LIN {X 0,Y 523.961,Z 128.215,A -85,B 0,C 180,E1 -4877.969,E2 -4877.969} C_VEL
LIN {X 0,Y 523.969,Z 128.221,A -85,B 0,C 180,E1 -4880.41,E2 -4880.41} C_VEL
LIN {X 0,Y 523.908,Z 128.222,A -85,B 0,C 180,E1 -4882.893,E2 -4882.893} C_VEL
LIN {X 0,Y 523.951,Z 128.214,A -85,B 0,C 180,E1 -4885.418,E2 -4885.418} C_VEL
LIN {X 0,Y 523.967,Z 128.217,A -85,B 0,C 180,E1 -4887.998,E2 -4887.998} C_VEL
LIN {X 0,Y 523.943,Z 128.216,A -85,B 0,C 180,E1 -4890.855,E2 -4890.855} C_VEL
LIN {X 0,Y 523.957,Z 128.217,A -85,B 0,C 180,E1 -4893.735,E2 -4893.735} C_VEL
LIN {X 0,Y 523.917,Z 128.223,A -85,B 0,C 180,E1 -4896.404,E2 -4896.404} C_VEL
LIN {X 0,Y 523.956,Z 128.214,A -85,B 0,C 180,E1 -4899.081,E2 -4899.081} C_VEL
LIN {X 0,Y 523.953,Z 128.221,A -85,B 0,C 180,E1 -4902.118,E2 -4902.118} C_VEL
LIN {X 0,Y 523.952,Z 128.216,A -85,B 0,C 180,E1 -4905.308,E2 -4905.308} C_VEL
LIN {X 0,Y 523.918,Z 128.218,A -85,B 0,C 180,E1 -4906.913,E2 -4906.913} C_VEL
LIN {X 0,Y 523.253,Z 128.307,A -85,B 0,C 180,E1 -4907.554,E2 -4907.554} C_VEL
LIN {X 0,Y 520.418,Z 128.661,A -85,B 0,C 180,E1 -4908.596,E2 -4908.596} C_VEL
LIN {X 0,Y 518.021,Z 128.96,A -85,B 0,C 180,E1 -4909.435,E2 -4909.435} C_VEL
LIN {X 0,Y 516.991,Z 129.087,A -85,B 0,C 180,E1 -4910.083,E2 -4910.083} C_VEL
LIN {X 0,Y 516.906,Z 129.094,A -85,B 0,C 180,E1 -4910.302,E2 -4910.302} C_VEL
LIN {X 0,Y 516.88,Z 129.098,A -85,B 0,C 180,E1 -4913.342,E2 -4913.342} C_VEL
LIN {X 0,Y 516.906,Z 129.095,A -85,B 0,C 180,E1 -4916.121,E2 -4916.121} C_VEL
LIN {X 0,Y 516.888,Z 129.095,A -85,B 0,C 180,E1 -4918.935,E2 -4918.935} C_VEL
LIN {X 0,Y 516.915,Z 129.1,A -85,B 0,C 180,E1 -4921.585,E2 -4921.585} C_VEL
LIN {X 0,Y 516.927,Z 129.09,A -85,B 0,C 180,E1 -4924.211,E2 -4924.211} C_VEL
LIN {X 0,Y 516.868,Z 129.097,A -85,B 0,C 180,E1 -4926.777,E2 -4926.777} C_VEL
LIN {X 0,Y 516.935,Z 129.093,A -85,B 0,C 180,E1 -4929.732,E2 -4929.732} C_VEL
LIN {X 0,Y 516.925,Z 129.09,A -85,B 0,C 180,E1 -4932.596,E2 -4932.596} C_VEL
LIN {X 0,Y 516.947,Z 129.092,A -85,B 0,C 180,E1 -4935.031,E2 -4935.031} C_VEL
LIN {X 0,Y 516.961,Z 129.085,A -85,B 0,C 180,E1 -4938.234,E2 -4938.234} C_VEL
LIN {X 0,Y 516.966,Z 129.09,A -85,B 0,C 180,E1 -4941.4,E2 -4941.4} C_VEL
LIN {X 0,Y 517.013,Z 129.08,A -85,B 0,C 180,E1 -4943.757,E2 -4943.757} C_VEL
LIN {X 0,Y 517.083,Z 129.071,A -85,B 0,C 180,E1 -4947.664,E2 -4947.664} C_VEL
LIN {X 0,Y 517.091,Z 129.075,A -85,B 0,C 180,E1 -4950.779,E2 -4950.779} C_VEL
LIN {X 0,Y 517.01,Z 129.085,A -85,B 0,C 180,E1 -4953.117,E2 -4953.117} C_VEL
LIN {X 0,Y 517.014,Z 129.08,A -85,B 0,C 180,E1 -4956.244,E2 -4956.244} C_VEL
LIN {X 0,Y 516.952,Z 129.088,A -85,B 0,C 180,E1 -4959.39,E2 -4959.39} C_VEL
LIN {X 0,Y 516.95,Z 129.086,A -85,B 0,C 180,E1 -4961.808,E2 -4961.808} C_VEL
LIN {X 0,Y 516.945,Z 129.092,A -85,B 0,C 180,E1 -4965.148,E2 -4965.148} C_VEL
LIN {X 0,Y 516.931,Z 129.096,A -85,B 0,C 180,E1 -4968.222,E2 -4968.222} C_VEL
LIN {X 0,Y 516.964,Z 129.166,A -85,B 0,C 180,E1 -4968.889,E2 -4968.889} C_VEL
LIN {X 0,Y 517.489,Z 133.922,A -85,B 0,C 180,E1 -4969.848,E2 -4969.848} C_VEL
LIN {X 0,Y 517.251,Z 148.414,A -85,B 0,C 180,E1 -4972.697,E2 -4972.697} C_VEL
LIN {X 0,Y 519.127,Z 158.271,A -85,B 0,C 180,E1 -4972.899,E2 -4972.899} C_VEL
LIN {X 0,Y 518.582,Z 255.219,A -85,B 0,C 180,E1 -4974.279,E2 -4974.279} C_VEL
LIN {X 0,Y 518.384,Z 268.208,A -85,B 0,C 180,E1 -4974.619,E2 -4974.619} C_VEL
LIN {X 0,Y 518.188,Z 281.309,A -85,B 0,C 180,E1 -4975.131,E2 -4975.131} C_VEL
LIN {X 0,Y 517.999,Z 292.599,A -85,B 0,C 180,E1 -4975.733,E2 -4975.733} C_VEL
LIN {X 0,Y 517.621,Z 304.359,A -85,B 0,C 180,E1 -4976.536,E2 -4976.536} C_VEL
LIN {X 0,Y 517.359,Z 314.43,A -85,B 0,C 180,E1 -4977.399,E2 -4977.399} C_VEL
LIN {X 0,Y 517.077,Z 323.966,A -85,B 0,C 180,E1 -4978.406,E2 -4978.406} C_VEL
LIN {X 0,Y 516.85,Z 332.431,A -85,B 0,C 180,E1 -4979.513,E2 -4979.513} C_VEL
LIN {X 0,Y 516.626,Z 340.432,A -85,B 0,C 180,E1 -4980.813,E2 -4980.813} C_VEL
LIN {X 0,Y 516.488,Z 346.396,A -85,B 0,C 180,E1 -4982.052,E2 -4982.052} C_VEL
LIN {X 0,Y 516.364,Z 351.459,A -85,B 0,C 180,E1 -4983.427,E2 -4983.427} C_VEL
LIN {X 0,Y 516.249,Z 355.267,A -85,B 0,C 180,E1 -4984.874,E2 -4984.874} C_VEL
LIN {X 0,Y 516.218,Z 356.939,A -85,B 0,C 180,E1 -4985.833,E2 -4985.833} C_VEL
LIN {X 0,Y 516.192,Z 358.058,A -85,B 0,C 180,E1 -4986.803,E2 -4986.803} C_VEL
LIN {X 0,Y 516.165,Z 358.528,A -85,B 0,C 180,E1 -4987.842,E2 -4987.842} C_VEL
LIN {X 0,Y 516.185,Z 358.189,A -85,B 0,C 180,E1 -4989.099,E2 -4989.099} C_VEL
LIN {X 0,Y 516.22,Z 356.867,A -85,B 0,C 180,E1 -4990.324,E2 -4990.324} C_VEL
LIN {X 0,Y 516.332,Z 353.874,A -85,B 0,C 180,E1 -4991.833,E2 -4991.833} C_VEL
LIN {X 0,Y 516.424,Z 349.132,A -85,B 0,C 180,E1 -4993.363,E2 -4993.363} C_VEL
LIN {X 0,Y 516.566,Z 343.421,A -85,B 0,C 180,E1 -4994.71,E2 -4994.71} C_VEL
LIN {X 0,Y 516.733,Z 337.42,A -85,B 0,C 180,E1 -4995.82,E2 -4995.82} C_VEL
LIN {X 0,Y 516.938,Z 329.156,A -85,B 0,C 180,E1 -4997.046,E2 -4997.046} C_VEL
LIN {X 0,Y 517.221,Z 320.09,A -85,B 0,C 180,E1 -4998.132,E2 -4998.132} C_VEL
LIN {X 0,Y 517.473,Z 310.551,A -85,B 0,C 180,E1 -4999.058,E2 -4999.058} C_VEL
LIN {X 0,Y 517.739,Z 300.481,A -85,B 0,C 180,E1 -4999.851,E2 -4999.851} C_VEL
LIN {X 0,Y 518.097,Z 289.313,A -85,B 0,C 180,E1 -5000.553,E2 -5000.553} C_VEL
LIN {X 0,Y 518.357,Z 276.664,A -85,B 0,C 180,E1 -5001.167,E2 -5001.167} C_VEL
LIN {X 0,Y 518.481,Z 264.053,A -85,B 0,C 180,E1 -5001.601,E2 -5001.601} C_VEL
LIN {X 0,Y 518.64,Z 250.833,A -85,B 0,C 180,E1 -5001.888,E2 -5001.888} C_VEL
LIN {X 0,Y 519.123,Z 157.894,A -85,B 0,C 180,E1 -5003.2,E2 -5003.2} C_VEL
LIN {X 0,Y 517.274,Z 148.573,A -85,B 0,C 180,E1 -5003.404,E2 -5003.404} C_VEL
LIN {X 0,Y 517.435,Z 134.125,A -85,B 0,C 180,E1 -5006.161,E2 -5006.161} C_VEL
LIN {X 0,Y 516.966,Z 129.093,A -85,B 0,C 180,E1 -5007.176,E2 -5007.176} C_VEL
LIN {X 0,Y 516.923,Z 129.093,A -85,B 0,C 180,E1 -5010.696,E2 -5010.696} C_VEL
LIN {X 0,Y 516.913,Z 129.096,A -85,B 0,C 180,E1 -5013.812,E2 -5013.812} C_VEL
LIN {X 0,Y 516.86,Z 129.105,A -85,B 0,C 180,E1 -5016.777,E2 -5016.777} C_VEL
LIN {X 0,Y 516.943,Z 129.09,A -85,B 0,C 180,E1 -5019.732,E2 -5019.732} C_VEL
LIN {X 0,Y 516.899,Z 129.099,A -85,B 0,C 180,E1 -5022.596,E2 -5022.596} C_VEL
LIN {X 0,Y 516.944,Z 129.095,A -85,B 0,C 180,E1 -5025.031,E2 -5025.031} C_VEL
LIN {X 0,Y 516.971,Z 129.089,A -85,B 0,C 180,E1 -5028.234,E2 -5028.234} C_VEL
LIN {X 0,Y 516.957,Z 129.088,A -85,B 0,C 180,E1 -5031.4,E2 -5031.4} C_VEL
LIN {X 0,Y 516.99,Z 129.089,A -85,B 0,C 180,E1 -5034.54,E2 -5034.54} C_VEL
LIN {X 0,Y 517.078,Z 129.073,A -85,B 0,C 180,E1 -5037.664,E2 -5037.664} C_VEL
LIN {X 0,Y 517.07,Z 129.075,A -85,B 0,C 180,E1 -5040,E2 -5040} C_VEL
LIN {X 0,Y 517.077,Z 129.075,A -85,B 0,C 180,E1 -5042.337,E2 -5042.337} C_VEL
LIN {X 0,Y 516.971,Z 129.086,A -85,B 0,C 180,E1 -5046.244,E2 -5046.244} C_VEL
LIN {X 0,Y 516.909,Z 129.094,A -85,B 0,C 180,E1 -5049.39,E2 -5049.39} C_VEL
LIN {X 0,Y 516.883,Z 129.095,A -85,B 0,C 180,E1 -5052.566,E2 -5052.566} C_VEL
LIN {X 0,Y 516.831,Z 129.107,A -85,B 0,C 180,E1 -5055.782,E2 -5055.782} C_VEL
LIN {X 0,Y 516.84,Z 129.101,A -85,B 0,C 180,E1 -5058.226,E2 -5058.226} C_VEL
LIN {X 0,Y 516.86,Z 129.098,A -85,B 0,C 180,E1 -5060.704,E2 -5060.704} C_VEL
LIN {X 0,Y 516.841,Z 129.107,A -85,B 0,C 180,E1 -5063.225,E2 -5063.225} C_VEL
LIN {X 0,Y 516.863,Z 129.098,A -85,B 0,C 180,E1 -5066.177,E2 -5066.177} C_VEL
LIN {X 0,Y 516.833,Z 129.1,A -85,B 0,C 180,E1 -5068.421,E2 -5068.421} C_VEL
LIN {X 0,Y 516.853,Z 129.105,A -85,B 0,C 180,E1 -5071.112,E2 -5071.112} C_VEL
LIN {X 0,Y 516.886,Z 129.095,A -85,B 0,C 180,E1 -5073.961,E2 -5073.961} C_VEL
LIN {X 0,Y 516.858,Z 129.105,A -85,B 0,C 180,E1 -5076.748,E2 -5076.748} C_VEL
LIN {X 0,Y 516.863,Z 129.099,A -85,B 0,C 180,E1 -5079.724,E2 -5079.724} C_VEL
LIN {X 0,Y 516.847,Z 129.107,A -85,B 0,C 180,E1 -5082.836,E2 -5082.836} C_VEL
LIN {X 0,Y 516.901,Z 129.098,A -85,B 0,C 180,E1 -5085.007,E2 -5085.007} C_VEL
LIN {X 0,Y 516.903,Z 129.102,A -85,B 0,C 180,E1 -5088.401,E2 -5088.401} C_VEL
LIN {X 0,Y 516.881,Z 129.097,A -85,B 0,C 180,E1 -5091.284,E2 -5091.284} C_VEL
LIN {X 0,Y 516.873,Z 129.105,A -85,B 0,C 180,E1 -5094.219,E2 -5094.219} C_VEL
LIN {X 0,Y 516.9,Z 129.097,A -85,B 0,C 180,E1 -5097.053,E2 -5097.053} C_VEL
LIN {X 0,Y 516.89,Z 129.102,A -85,B 0,C 180,E1 -5099.796,E2 -5099.796} C_VEL
LIN {X 0,Y 516.904,Z 129.098,A -85,B 0,C 180,E1 -5102.465,E2 -5102.465} C_VEL
LIN {X 0,Y 516.94,Z 129.172,A -85,B 0,C 180,E1 -5105.019,E2 -5105.019} C_VEL
LIN {X 0,Y 518.404,Z 137.817,A -85,B 0,C 180,E1 -5106.426,E2 -5106.426} C_VEL
LIN {X 0,Y 517.908,Z 158.298,A -85,B 0,C 180,E1 -5109.545,E2 -5109.545} C_VEL
LIN {X 0,Y 517.54,Z 177.537,A -85,B 0,C 180,E1 -5112.439,E2 -5112.439} C_VEL
LIN {X 0,Y 517.196,Z 192.388,A -85,B 0,C 180,E1 -5114.631,E2 -5114.631} C_VEL
LIN {X 0,Y 519.037,Z 206.215,A -85,B 0,C 180,E1 -5114.883,E2 -5114.883} C_VEL
LIN {X 0,Y 518.573,Z 300.986,A -85,B 0,C 180,E1 -5116.23,E2 -5116.23} C_VEL
LIN {X 0,Y 518.317,Z 314.244,A -85,B 0,C 180,E1 -5116.573,E2 -5116.573} C_VEL
LIN {X 0,Y 518.011,Z 326.993,A -85,B 0,C 180,E1 -5117.064,E2 -5117.064} C_VEL
LIN {X 0,Y 517.751,Z 338.84,A -85,B 0,C 180,E1 -5117.686,E2 -5117.686} C_VEL
LIN {X 0,Y 517.454,Z 350.053,A -85,B 0,C 180,E1 -5118.443,E2 -5118.443} C_VEL
LIN {X 0,Y 517.162,Z 360.598,A -85,B 0,C 180,E1 -5119.329,E2 -5119.329} C_VEL
LIN {X 0,Y 516.896,Z 369.22,A -85,B 0,C 180,E1 -5120.214,E2 -5120.214} C_VEL
LIN {X 0,Y 516.68,Z 377.176,A -85,B 0,C 180,E1 -5121.197,E2 -5121.197} C_VEL
LIN {X 0,Y 516.516,Z 384.949,A -85,B 0,C 180,E1 -5122.376,E2 -5122.376} C_VEL
LIN {X 0,Y 516.376,Z 392.107,A -85,B 0,C 180,E1 -5123.749,E2 -5123.749} C_VEL
LIN {X 0,Y 516.312,Z 396.873,A -85,B 0,C 180,E1 -5124.924,E2 -5124.924} C_VEL
LIN {X 0,Y 516.352,Z 400.52,A -85,B 0,C 180,E1 -5126.097,E2 -5126.097} C_VEL
LIN {X 0,Y 516.303,Z 402.399,A -85,B 0,C 180,E1 -5126.878,E2 -5126.878} C_VEL
LIN {X 0,Y 516.264,Z 403.807,A -85,B 0,C 180,E1 -5127.659,E2 -5127.659} C_VEL
LIN {X 0,Y 516.172,Z 405.428,A -85,B 0,C 180,E1 -5129.219,E2 -5129.219} C_VEL
LIN {X 0,Y 516.173,Z 405.651,A -85,B 0,C 180,E1 -5130,E2 -5130} C_VEL
LIN {X 0,Y 516.193,Z 404.83,A -85,B 0,C 180,E1 -5131.56,E2 -5131.56} C_VEL
LIN {X 0,Y 516.264,Z 403.836,A -85,B 0,C 180,E1 -5132.34,E2 -5132.34} C_VEL
LIN {X 0,Y 516.303,Z 402.435,A -85,B 0,C 180,E1 -5133.121,E2 -5133.121} C_VEL
LIN {X 0,Y 516.31,Z 399.485,A -85,B 0,C 180,E1 -5134.293,E2 -5134.293} C_VEL
LIN {X 0,Y 516.367,Z 395.491,A -85,B 0,C 180,E1 -5135.467,E2 -5135.467} C_VEL
LIN {X 0,Y 516.41,Z 390.303,A -85,B 0,C 180,E1 -5136.651,E2 -5136.651} C_VEL
LIN {X 0,Y 516.534,Z 383.867,A -85,B 0,C 180,E1 -5137.82,E2 -5137.82} C_VEL
LIN {X 0,Y 516.741,Z 375.791,A -85,B 0,C 180,E1 -5138.998,E2 -5138.998} C_VEL
LIN {X 0,Y 516.93,Z 367.556,A -85,B 0,C 180,E1 -5139.982,E2 -5139.982} C_VEL
LIN {X 0,Y 517.224,Z 357.517,A -85,B 0,C 180,E1 -5140.966,E2 -5140.966} C_VEL
LIN {X 0,Y 517.504,Z 347.593,A -85,B 0,C 180,E1 -5141.753,E2 -5141.753} C_VEL
LIN {X 0,Y 517.83,Z 336.445,A -85,B 0,C 180,E1 -5142.462,E2 -5142.462} C_VEL
LIN {X 0,Y 518.108,Z 323.829,A -85,B 0,C 180,E1 -5143.083,E2 -5143.083} C_VEL
LIN {X 0,Y 518.408,Z 311.414,A -85,B 0,C 180,E1 -5143.524,E2 -5143.524} C_VEL
LIN {X 0,Y 518.607,Z 298.558,A -85,B 0,C 180,E1 -5143.818,E2 -5143.818} C_VEL
LIN {X 0,Y 518.962,Z 204.412,A -85,B 0,C 180,E1 -5145.149,E2 -5145.149} C_VEL
LIN {X 0,Y 517.228,Z 192.469,A -85,B 0,C 180,E1 -5145.389,E2 -5145.389} C_VEL
LIN {X 0,Y 517.694,Z 172.47,A -85,B 0,C 180,E1 -5148.399,E2 -5148.399} C_VEL
LIN {X 0,Y 518.188,Z 152.265,A -85,B 0,C 180,E1 -5151.48,E2 -5151.48} C_VEL
LIN {X 0,Y 518.583,Z 138.788,A -85,B 0,C 180,E1 -5153.565,E2 -5153.565} C_VEL
LIN {X 0,Y 517.236,Z 130.625,A -85,B 0,C 180,E1 -5154.911,E2 -5154.911} C_VEL
LIN {X 0,Y 516.922,Z 129.096,A -85,B 0,C 180,E1 -5155.196,E2 -5155.196} C_VEL
LIN {X 0,Y 516.917,Z 129.098,A -85,B 0,C 180,E1 -5157.903,E2 -5157.903} C_VEL
LIN {X 0,Y 516.893,Z 129.101,A -85,B 0,C 180,E1 -5160.203,E2 -5160.203} C_VEL
LIN {X 0,Y 516.896,Z 129.093,A -85,B 0,C 180,E1 -5162.946,E2 -5162.946} C_VEL
LIN {X 0,Y 516.871,Z 129.103,A -85,B 0,C 180,E1 -5165.78,E2 -5165.78} C_VEL
LIN {X 0,Y 516.882,Z 129.095,A -85,B 0,C 180,E1 -5168.715,E2 -5168.715} C_VEL
LIN {X 0,Y 516.912,Z 129.099,A -85,B 0,C 180,E1 -5171.775,E2 -5171.775} C_VEL
LIN {X 0,Y 516.895,Z 129.094,A -85,B 0,C 180,E1 -5175.006,E2 -5175.006} C_VEL
LIN {X 0,Y 516.915,Z 129.091,A -85,B 0,C 180,E1 -5178.398,E2 -5178.398} C_VEL
LIN {X 0,Y 516.88,Z 129.099,A -85,B 0,C 180,E1 -5181.284,E2 -5181.284} C_VEL
LIN {X 0,Y 516.87,Z 129.097,A -85,B 0,C 180,E1 -5184.219,E2 -5184.219} C_VEL
LIN {X 0,Y 516.88,Z 129.098,A -85,B 0,C 180,E1 -5187.052,E2 -5187.052} C_VEL
LIN {X 0,Y 516.886,Z 129.098,A -85,B 0,C 180,E1 -5189.796,E2 -5189.796} C_VEL
LIN {X 0,Y 516.925,Z 129.089,A -85,B 0,C 180,E1 -5192.467,E2 -5192.467} C_VEL
LIN {X 0,Y 516.908,Z 129.096,A -85,B 0,C 180,E1 -5195.071,E2 -5195.071} C_VEL
LIN {X 0,Y 516.885,Z 129.095,A -85,B 0,C 180,E1 -5198.462,E2 -5198.462} C_VEL
LIN {X 0,Y 516.899,Z 129.098,A -85,B 0,C 180,E1 -5200.954,E2 -5200.954} C_VEL
LIN {X 0,Y 516.907,Z 129.097,A -85,B 0,C 180,E1 -5203.41,E2 -5203.41} C_VEL
LIN {X 0,Y 516.893,Z 129.094,A -85,B 0,C 180,E1 -5205.833,E2 -5205.833} C_VEL
LIN {X 0,Y 516.965,Z 129.085,A -85,B 0,C 180,E1 -5208.233,E2 -5208.233} C_VEL
LIN {X 0,Y 516.967,Z 129.088,A -85,B 0,C 180,E1 -5211.399,E2 -5211.399} C_VEL
LIN {X 0,Y 517.002,Z 129.08,A -85,B 0,C 180,E1 -5213.756,E2 -5213.756} C_VEL
LIN {X 0,Y 517.012,Z 129.088,A -85,B 0,C 180,E1 -5216.883,E2 -5216.883} C_VEL
LIN {X 0,Y 517.084,Z 129.07,A -85,B 0,C 180,E1 -5220,E2 -5220} C_VEL
LIN {X 0,Y 517.01,Z 129.083,A -85,B 0,C 180,E1 -5223.117,E2 -5223.117} C_VEL
LIN {X 0,Y 517.001,Z 129.083,A -85,B 0,C 180,E1 -5226.243,E2 -5226.243} C_VEL
LIN {X 0,Y 516.952,Z 129.087,A -85,B 0,C 180,E1 -5229.389,E2 -5229.389} C_VEL
LIN {X 0,Y 516.95,Z 129.087,A -85,B 0,C 180,E1 -5231.807,E2 -5231.807} C_VEL
LIN {X 0,Y 516.944,Z 129.088,A -85,B 0,C 180,E1 -5235.147,E2 -5235.147} C_VEL
LIN {X 0,Y 516.922,Z 129.095,A -85,B 0,C 180,E1 -5238.222,E2 -5238.222} C_VEL
LIN {X 0,Y 516.909,Z 129.096,A -85,B 0,C 180,E1 -5240.701,E2 -5240.701} C_VEL
LIN {X 0,Y 516.9,Z 129.097,A -85,B 0,C 180,E1 -5244.072,E2 -5244.072} C_VEL
LIN {X 0,Y 516.926,Z 129.093,A -85,B 0,C 180,E1 -5246.657,E2 -5246.657} C_VEL
LIN {X 0,Y 516.908,Z 129.092,A -85,B 0,C 180,E1 -5249.524,E2 -5249.524} C_VEL
LIN {X 0,Y 516.897,Z 129.097,A -85,B 0,C 180,E1 -5252.544,E2 -5252.544} C_VEL
LIN {X 0,Y 516.876,Z 129.096,A -85,B 0,C 180,E1 -5255.332,E2 -5255.332} C_VEL
LIN {X 0,Y 516.878,Z 129.103,A -85,B 0,C 180,E1 -5257.943,E2 -5257.943} C_VEL
LIN {X 0,Y 516.9,Z 129.093,A -85,B 0,C 180,E1 -5260.739,E2 -5260.739} C_VEL
LIN {X 0,Y 516.878,Z 129.104,A -85,B 0,C 180,E1 -5263.903,E2 -5263.903} C_VEL
LIN {X 0,Y 516.878,Z 129.101,A -85,B 0,C 180,E1 -5266.107,E2 -5266.107} C_VEL
LIN {X 0,Y 516.899,Z 129.094,A -85,B 0,C 180,E1 -5269.26,E2 -5269.26} C_VEL
LIN {X 0,Y 516.906,Z 129.094,A -85,B 0,C 180,E1 -5270.302,E2 -5270.302} C_VEL
LIN {X 0,Y 516.237,Z 129.176,A -85,B 0,C 180,E1 -5270.952,E2 -5270.952} C_VEL
LIN {X 0,Y 513.38,Z 129.538,A -85,B 0,C 180,E1 -5272.007,E2 -5272.007} C_VEL
LIN {X 0,Y 510.961,Z 129.844,A -85,B 0,C 180,E1 -5272.857,E2 -5272.857} C_VEL
LIN {X 0,Y 509.915,Z 129.972,A -85,B 0,C 180,E1 -5273.514,E2 -5273.514} C_VEL
LIN {X 0,Y 509.826,Z 129.98,A -85,B 0,C 180,E1 -5273.736,E2 -5273.736} C_VEL
LIN {X 0,Y 509.857,Z 129.97,A -85,B 0,C 180,E1 -5276.539,E2 -5276.539} C_VEL
LIN {X 0,Y 509.841,Z 129.976,A -85,B 0,C 180,E1 -5279.334,E2 -5279.334} C_VEL
LIN {X 0,Y 509.89,Z 129.968,A -85,B 0,C 180,E1 -5282.055,E2 -5282.055} C_VEL
LIN {X 0,Y 509.873,Z 129.968,A -85,B 0,C 180,E1 -5284.704,E2 -5284.704} C_VEL
LIN {X 0,Y 509.852,Z 129.98,A -85,B 0,C 180,E1 -5287.45,E2 -5287.45} C_VEL
LIN {X 0,Y 509.913,Z 129.966,A -85,B 0,C 180,E1 -5289.845,E2 -5289.845} C_VEL
LIN {X 0,Y 509.881,Z 129.973,A -85,B 0,C 180,E1 -5293.175,E2 -5293.175} C_VEL
LIN {X 0,Y 509.869,Z 129.972,A -85,B 0,C 180,E1 -5295.635,E2 -5295.635} C_VEL
LIN {X 0,Y 509.91,Z 129.967,A -85,B 0,C 180,E1 -5298.875,E2 -5298.875} C_VEL
LIN {X 0,Y 509.948,Z 129.959,A -85,B 0,C 180,E1 -5302.079,E2 -5302.079} C_VEL
LIN {X 0,Y 509.983,Z 129.955,A -85,B 0,C 180,E1 -5304.465,E2 -5304.465} C_VEL
LIN {X 0,Y 510.054,Z 129.947,A -85,B 0,C 180,E1 -5307.631,E2 -5307.631} C_VEL
LIN {X 0,Y 510.061,Z 129.951,A -85,B 0,C 180,E1 -5310.79,E2 -5310.79} C_VEL
LIN {X 0,Y 509.952,Z 129.964,A -85,B 0,C 180,E1 -5313.161,E2 -5313.161} C_VEL
LIN {X 0,Y 509.981,Z 129.956,A -85,B 0,C 180,E1 -5316.33,E2 -5316.33} C_VEL
LIN {X 0,Y 509.914,Z 129.97,A -85,B 0,C 180,E1 -5318.721,E2 -5318.721} C_VEL
LIN {X 0,Y 509.902,Z 129.965,A -85,B 0,C 180,E1 -5321.932,E2 -5321.932} C_VEL
LIN {X 0,Y 509.892,Z 129.97,A -85,B 0,C 180,E1 -5325.242,E2 -5325.242} C_VEL
LIN {X 0,Y 509.883,Z 129.976,A -85,B 0,C 180,E1 -5328.483,E2 -5328.483} C_VEL
LIN {X 0,Y 509.945,Z 130.203,A -85,B 0,C 180,E1 -5328.794,E2 -5328.794} C_VEL
LIN {X 0,Y 510.5,Z 135.748,A -85,B 0,C 180,E1 -5329.922,E2 -5329.922} C_VEL
LIN {X 0,Y 510.268,Z 148.653,A -85,B 0,C 180,E1 -5332.48,E2 -5332.48} C_VEL
LIN {X 0,Y 512.304,Z 159.447,A -85,B 0,C 180,E1 -5332.706,E2 -5332.706} C_VEL
LIN {X 0,Y 511.687,Z 256.025,A -85,B 0,C 180,E1 -5334.105,E2 -5334.105} C_VEL
LIN {X 0,Y 511.49,Z 269.228,A -85,B 0,C 180,E1 -5334.462,E2 -5334.462} C_VEL
LIN {X 0,Y 511.297,Z 281.411,A -85,B 0,C 180,E1 -5334.948,E2 -5334.948} C_VEL
LIN {X 0,Y 511.071,Z 292.81,A -85,B 0,C 180,E1 -5335.56,E2 -5335.56} C_VEL
LIN {X 0,Y 510.738,Z 303.116,A -85,B 0,C 180,E1 -5336.261,E2 -5336.261} C_VEL
LIN {X 0,Y 510.416,Z 313.477,A -85,B 0,C 180,E1 -5337.136,E2 -5337.136} C_VEL
LIN {X 0,Y 510.097,Z 323.155,A -85,B 0,C 180,E1 -5338.144,E2 -5338.144} C_VEL
LIN {X 0,Y 509.847,Z 332.075,A -85,B 0,C 180,E1 -5339.298,E2 -5339.298} C_VEL
LIN {X 0,Y 509.636,Z 339.27,A -85,B 0,C 180,E1 -5340.451,E2 -5340.451} C_VEL
LIN {X 0,Y 509.461,Z 345.149,A -85,B 0,C 180,E1 -5341.616,E2 -5341.616} C_VEL
LIN {X 0,Y 509.307,Z 350.833,A -85,B 0,C 180,E1 -5343.063,E2 -5343.063} C_VEL
LIN {X 0,Y 509.203,Z 354.759,A -85,B 0,C 180,E1 -5344.464,E2 -5344.464} C_VEL
LIN {X 0,Y 509.132,Z 356.774,A -85,B 0,C 180,E1 -5345.47,E2 -5345.47} C_VEL
LIN {X 0,Y 509.1,Z 358.394,A -85,B 0,C 180,E1 -5346.806,E2 -5346.806} C_VEL
LIN {X 0,Y 509.083,Z 358.882,A -85,B 0,C 180,E1 -5348.104,E2 -5348.104} C_VEL
LIN {X 0,Y 509.114,Z 358.288,A -85,B 0,C 180,E1 -5349.421,E2 -5349.421} C_VEL
LIN {X 0,Y 509.156,Z 356.823,A -85,B 0,C 180,E1 -5350.609,E2 -5350.609} C_VEL
LIN {X 0,Y 509.263,Z 354.358,A -85,B 0,C 180,E1 -5351.823,E2 -5351.823} C_VEL
LIN {X 0,Y 509.345,Z 350.01,A -85,B 0,C 180,E1 -5353.28,E2 -5353.28} C_VEL
LIN {X 0,Y 509.495,Z 344.178,A -85,B 0,C 180,E1 -5354.709,E2 -5354.709} C_VEL
LIN {X 0,Y 509.68,Z 338.416,A -85,B 0,C 180,E1 -5355.811,E2 -5355.811} C_VEL
LIN {X 0,Y 509.854,Z 331.216,A -85,B 0,C 180,E1 -5356.935,E2 -5356.935} C_VEL
LIN {X 0,Y 510.159,Z 322.216,A -85,B 0,C 180,E1 -5358.066,E2 -5358.066} C_VEL
LIN {X 0,Y 510.486,Z 311.835,A -85,B 0,C 180,E1 -5359.121,E2 -5359.121} C_VEL
LIN {X 0,Y 510.763,Z 301.309,A -85,B 0,C 180,E1 -5359.976,E2 -5359.976} C_VEL
LIN {X 0,Y 511.141,Z 290.511,A -85,B 0,C 180,E1 -5360.674,E2 -5360.674} C_VEL
LIN {X 0,Y 511.403,Z 278.832,A -85,B 0,C 180,E1 -5361.263,E2 -5361.263} C_VEL
LIN {X 0,Y 511.58,Z 266.201,A -85,B 0,C 180,E1 -5361.732,E2 -5361.732} C_VEL
LIN {X 0,Y 511.718,Z 253.647,A -85,B 0,C 180,E1 -5362.034,E2 -5362.034} C_VEL
LIN {X 0,Y 512.294,Z 158.765,A -85,B 0,C 180,E1 -5363.4,E2 -5363.4} C_VEL
LIN {X 0,Y 510.314,Z 148.809,A -85,B 0,C 180,E1 -5363.631,E2 -5363.631} C_VEL
LIN {X 0,Y 510.453,Z 134.587,A -85,B 0,C 180,E1 -5366.361,E2 -5366.361} C_VEL
LIN {X 0,Y 509.906,Z 129.973,A -85,B 0,C 180,E1 -5367.292,E2 -5367.292} C_VEL
LIN {X 0,Y 509.86,Z 129.972,A -85,B 0,C 180,E1 -5370.275,E2 -5370.275} C_VEL
LIN {X 0,Y 509.878,Z 129.975,A -85,B 0,C 180,E1 -5372.945,E2 -5372.945} C_VEL
LIN {X 0,Y 509.843,Z 129.978,A -85,B 0,C 180,E1 -5375.573,E2 -5375.573} C_VEL
LIN {X 0,Y 509.824,Z 129.977,A -85,B 0,C 180,E1 -5378.149,E2 -5378.149} C_VEL
LIN {X 0,Y 509.86,Z 129.976,A -85,B 0,C 180,E1 -5380.682,E2 -5380.682} C_VEL
LIN {X 0,Y 509.867,Z 129.975,A -85,B 0,C 180,E1 -5383.175,E2 -5383.175} C_VEL
LIN {X 0,Y 509.858,Z 129.973,A -85,B 0,C 180,E1 -5385.634,E2 -5385.634} C_VEL
LIN {X 0,Y 509.916,Z 129.969,A -85,B 0,C 180,E1 -5388.875,E2 -5388.875} C_VEL
LIN {X 0,Y 509.912,Z 129.968,A -85,B 0,C 180,E1 -5392.078,E2 -5392.078} C_VEL
LIN {X 0,Y 509.945,Z 129.968,A -85,B 0,C 180,E1 -5394.464,E2 -5394.464} C_VEL
LIN {X 0,Y 510.046,Z 129.949,A -85,B 0,C 180,E1 -5397.631,E2 -5397.631} C_VEL
LIN {X 0,Y 510.038,Z 129.951,A -85,B 0,C 180,E1 -5400,E2 -5400} C_VEL
LIN {X 0,Y 510.045,Z 129.95,A -85,B 0,C 180,E1 -5402.37,E2 -5402.37} C_VEL
LIN {X 0,Y 509.939,Z 129.963,A -85,B 0,C 180,E1 -5405.537,E2 -5405.537} C_VEL
LIN {X 0,Y 509.879,Z 129.973,A -85,B 0,C 180,E1 -5407.923,E2 -5407.923} C_VEL
LIN {X 0,Y 509.864,Z 129.967,A -85,B 0,C 180,E1 -5411.127,E2 -5411.127} C_VEL
LIN {X 0,Y 509.815,Z 129.981,A -85,B 0,C 180,E1 -5413.554,E2 -5413.554} C_VEL
LIN {X 0,Y 509.792,Z 129.982,A -85,B 0,C 180,E1 -5416.005,E2 -5416.005} C_VEL
LIN {X 0,Y 509.806,Z 129.976,A -85,B 0,C 180,E1 -5418.486,E2 -5418.486} C_VEL
LIN {X 0,Y 509.812,Z 129.978,A -85,B 0,C 180,E1 -5421.004,E2 -5421.004} C_VEL
LIN {X 0,Y 509.802,Z 129.981,A -85,B 0,C 180,E1 -5423.565,E2 -5423.565} C_VEL
LIN {X 0,Y 509.804,Z 129.977,A -85,B 0,C 180,E1 -5426.353,E2 -5426.353} C_VEL
LIN {X 0,Y 509.797,Z 129.98,A -85,B 0,C 180,E1 -5428.85,E2 -5428.85} C_VEL
LIN {X 0,Y 509.801,Z 129.979,A -85,B 0,C 180,E1 -5431.592,E2 -5431.592} C_VEL
LIN {X 0,Y 509.839,Z 129.975,A -85,B 0,C 180,E1 -5434.415,E2 -5434.415} C_VEL
LIN {X 0,Y 509.812,Z 129.978,A -85,B 0,C 180,E1 -5437.342,E2 -5437.342} C_VEL
LIN {X 0,Y 509.819,Z 129.979,A -85,B 0,C 180,E1 -5440.385,E2 -5440.385} C_VEL
LIN {X 0,Y 509.81,Z 129.977,A -85,B 0,C 180,E1 -5443.573,E2 -5443.573} C_VEL
LIN {X 0,Y 509.813,Z 129.984,A -85,B 0,C 180,E1 -5446.427,E2 -5446.427} C_VEL
LIN {X 0,Y 509.826,Z 129.977,A -85,B 0,C 180,E1 -5449.305,E2 -5449.305} C_VEL
LIN {X 0,Y 509.854,Z 129.974,A -85,B 0,C 180,E1 -5451.787,E2 -5451.787} C_VEL
LIN {X 0,Y 509.832,Z 129.978,A -85,B 0,C 180,E1 -5454.622,E2 -5454.622} C_VEL
LIN {X 0,Y 509.866,Z 129.974,A -85,B 0,C 180,E1 -5457.481,E2 -5457.481} C_VEL
LIN {X 0,Y 509.863,Z 129.977,A -85,B 0,C 180,E1 -5460.274,E2 -5460.274} C_VEL
LIN {X 0,Y 509.884,Z 129.974,A -85,B 0,C 180,E1 -5463.629,E2 -5463.629} C_VEL
LIN {X 0,Y 509.888,Z 129.999,A -85,B 0,C 180,E1 -5464.838,E2 -5464.838} C_VEL
LIN {X 0,Y 511.457,Z 138.841,A -85,B 0,C 180,E1 -5466.301,E2 -5466.301} C_VEL
LIN {X 0,Y 510.986,Z 158.737,A -85,B 0,C 180,E1 -5469.378,E2 -5469.378} C_VEL
LIN {X 0,Y 510.526,Z 178.372,A -85,B 0,C 180,E1 -5472.37,E2 -5472.37} C_VEL
LIN {X 0,Y 510.198,Z 191.955,A -85,B 0,C 180,E1 -5474.413,E2 -5474.413} C_VEL
LIN {X 0,Y 512.182,Z 206.713,A -85,B 0,C 180,E1 -5474.689,E2 -5474.689} C_VEL
LIN {X 0,Y 511.683,Z 300.481,A -85,B 0,C 180,E1 -5476.041,E2 -5476.041} C_VEL
LIN {X 0,Y 511.395,Z 313.787,A -85,B 0,C 180,E1 -5476.388,E2 -5476.388} C_VEL
LIN {X 0,Y 511.071,Z 326.562,A -85,B 0,C 180,E1 -5476.885,E2 -5476.885} C_VEL
LIN {X 0,Y 510.77,Z 338.533,A -85,B 0,C 180,E1 -5477.521,E2 -5477.521} C_VEL
LIN {X 0,Y 510.448,Z 349.663,A -85,B 0,C 180,E1 -5478.282,E2 -5478.282} C_VEL
LIN {X 0,Y 510.15,Z 360.22,A -85,B 0,C 180,E1 -5479.181,E2 -5479.181} C_VEL
LIN {X 0,Y 509.835,Z 368.849,A -85,B 0,C 180,E1 -5480.077,E2 -5480.077} C_VEL
LIN {X 0,Y 509.64,Z 376.815,A -85,B 0,C 180,E1 -5481.075,E2 -5481.075} C_VEL
LIN {X 0,Y 509.429,Z 384.596,A -85,B 0,C 180,E1 -5482.269,E2 -5482.269} C_VEL
LIN {X 0,Y 509.31,Z 390.938,A -85,B 0,C 180,E1 -5483.483,E2 -5483.483} C_VEL
LIN {X 0,Y 509.241,Z 396.536,A -85,B 0,C 180,E1 -5484.853,E2 -5484.853} C_VEL
LIN {X 0,Y 509.246,Z 400.186,A -85,B 0,C 180,E1 -5486.043,E2 -5486.043} C_VEL
LIN {X 0,Y 509.219,Z 402.069,A -85,B 0,C 180,E1 -5486.835,E2 -5486.835} C_VEL
LIN {X 0,Y 509.193,Z 403.48,A -85,B 0,C 180,E1 -5487.626,E2 -5487.626} C_VEL
LIN {X 0,Y 509.085,Z 405.104,A -85,B 0,C 180,E1 -5489.209,E2 -5489.209} C_VEL
LIN {X 0,Y 509.083,Z 405.328,A -85,B 0,C 180,E1 -5490,E2 -5490} C_VEL
LIN {X 0,Y 509.113,Z 404.509,A -85,B 0,C 180,E1 -5491.582,E2 -5491.582} C_VEL
LIN {X 0,Y 509.193,Z 403.514,A -85,B 0,C 180,E1 -5492.373,E2 -5492.373} C_VEL
LIN {X 0,Y 509.219,Z 402.112,A -85,B 0,C 180,E1 -5493.164,E2 -5493.164} C_VEL
LIN {X 0,Y 509.203,Z 399.16,A -85,B 0,C 180,E1 -5494.353,E2 -5494.353} C_VEL
LIN {X 0,Y 509.279,Z 395.164,A -85,B 0,C 180,E1 -5495.543,E2 -5495.543} C_VEL
LIN {X 0,Y 509.366,Z 389.113,A -85,B 0,C 180,E1 -5496.914,E2 -5496.914} C_VEL
LIN {X 0,Y 509.493,Z 382.289,A -85,B 0,C 180,E1 -5498.128,E2 -5498.128} C_VEL
LIN {X 0,Y 509.715,Z 373.952,A -85,B 0,C 180,E1 -5499.323,E2 -5499.323} C_VEL
LIN {X 0,Y 509.957,Z 365.393,A -85,B 0,C 180,E1 -5500.32,E2 -5500.32} C_VEL
LIN {X 0,Y 510.328,Z 354.826,A -85,B 0,C 180,E1 -5501.317,E2 -5501.317} C_VEL
LIN {X 0,Y 510.584,Z 344.031,A -85,B 0,C 180,E1 -5502.14,E2 -5502.14} C_VEL
LIN {X 0,Y 510.934,Z 332.88,A -85,B 0,C 180,E1 -5502.814,E2 -5502.814} C_VEL
LIN {X 0,Y 511.218,Z 321.009,A -85,B 0,C 180,E1 -5503.363,E2 -5503.363} C_VEL
LIN {X 0,Y 511.529,Z 307.326,A -85,B 0,C 180,E1 -5503.81,E2 -5503.81} C_VEL
LIN {X 0,Y 511.754,Z 295.057,A -85,B 0,C 180,E1 -5504.058,E2 -5504.058} C_VEL
LIN {X 0,Y 511.999,Z 204.354,A -85,B 0,C 180,E1 -5505.356,E2 -5505.356} C_VEL
LIN {X 0,Y 510.208,Z 192.178,A -85,B 0,C 180,E1 -5505.603,E2 -5505.603} C_VEL
LIN {X 0,Y 510.752,Z 170.815,A -85,B 0,C 180,E1 -5508.866,E2 -5508.866} C_VEL
LIN {X 0,Y 511.358,Z 149.282,A -85,B 0,C 180,E1 -5512.207,E2 -5512.207} C_VEL
LIN {X 0,Y 511.528,Z 138.482,A -85,B 0,C 180,E1 -5513.91,E2 -5513.91} C_VEL
LIN {X 0,Y 509.874,Z 129.975,A -85,B 0,C 180,E1 -5515.35,E2 -5515.35} C_VEL
LIN {X 0,Y 509.89,Z 129.974,A -85,B 0,C 180,E1 -5518.098,E2 -5518.098} C_VEL
LIN {X 0,Y 509.847,Z 129.972,A -85,B 0,C 180,E1 -5521.279,E2 -5521.279} C_VEL
LIN {X 0,Y 509.857,Z 129.976,A -85,B 0,C 180,E1 -5524.202,E2 -5524.202} C_VEL
LIN {X 0,Y 509.817,Z 129.976,A -85,B 0,C 180,E1 -5527.34,E2 -5527.34} C_VEL
LIN {X 0,Y 509.838,Z 129.974,A -85,B 0,C 180,E1 -5530.382,E2 -5530.382} C_VEL
LIN {X 0,Y 509.822,Z 129.975,A -85,B 0,C 180,E1 -5533.062,E2 -5533.062} C_VEL
LIN {X 0,Y 509.823,Z 129.983,A -85,B 0,C 180,E1 -5535.793,E2 -5535.793} C_VEL
LIN {X 0,Y 509.857,Z 129.97,A -85,B 0,C 180,E1 -5538.574,E2 -5538.574} C_VEL
LIN {X 0,Y 509.851,Z 129.977,A -85,B 0,C 180,E1 -5541.786,E2 -5541.786} C_VEL
LIN {X 0,Y 509.829,Z 129.973,A -85,B 0,C 180,E1 -5544.621,E2 -5544.621} C_VEL
LIN {X 0,Y 509.859,Z 129.978,A -85,B 0,C 180,E1 -5547.48,E2 -5547.48} C_VEL
LIN {X 0,Y 509.857,Z 129.97,A -85,B 0,C 180,E1 -5550.273,E2 -5550.273} C_VEL
LIN {X 0,Y 509.883,Z 129.969,A -85,B 0,C 180,E1 -5552.944,E2 -5552.944} C_VEL
LIN {X 0,Y 509.864,Z 129.975,A -85,B 0,C 180,E1 -5555.573,E2 -5555.573} C_VEL
LIN {X 0,Y 509.849,Z 129.976,A -85,B 0,C 180,E1 -5558.998,E2 -5558.998} C_VEL
LIN {X 0,Y 509.86,Z 129.974,A -85,B 0,C 180,E1 -5561.516,E2 -5561.516} C_VEL
LIN {X 0,Y 509.852,Z 129.971,A -85,B 0,C 180,E1 -5563.997,E2 -5563.997} C_VEL
LIN {X 0,Y 509.861,Z 129.97,A -85,B 0,C 180,E1 -5566.447,E2 -5566.447} C_VEL
LIN {X 0,Y 509.912,Z 129.969,A -85,B 0,C 180,E1 -5568.874,E2 -5568.874} C_VEL
LIN {X 0,Y 509.95,Z 129.958,A -85,B 0,C 180,E1 -5572.078,E2 -5572.078} C_VEL
LIN {X 0,Y 509.979,Z 129.957,A -85,B 0,C 180,E1 -5574.464,E2 -5574.464} C_VEL
LIN {X 0,Y 510.055,Z 129.946,A -85,B 0,C 180,E1 -5577.63,E2 -5577.63} C_VEL
LIN {X 0,Y 510.063,Z 129.953,A -85,B 0,C 180,E1 -5580.789,E2 -5580.789} C_VEL
LIN {X 0,Y 509.952,Z 129.962,A -85,B 0,C 180,E1 -5583.16,E2 -5583.16} C_VEL
LIN {X 0,Y 509.953,Z 129.962,A -85,B 0,C 180,E1 -5586.329,E2 -5586.329} C_VEL
LIN {X 0,Y 509.914,Z 129.971,A -85,B 0,C 180,E1 -5588.72,E2 -5588.72} C_VEL
LIN {X 0,Y 509.902,Z 129.965,A -85,B 0,C 180,E1 -5591.931,E2 -5591.931} C_VEL
LIN {X 0,Y 509.891,Z 129.966,A -85,B 0,C 180,E1 -5595.241,E2 -5595.241} C_VEL
LIN {X 0,Y 509.886,Z 129.969,A -85,B 0,C 180,E1 -5598.001,E2 -5598.001} C_VEL
LIN {X 0,Y 509.847,Z 129.973,A -85,B 0,C 180,E1 -5601.001,E2 -5601.001} C_VEL
LIN {X 0,Y 509.862,Z 129.977,A -85,B 0,C 180,E1 -5604.426,E2 -5604.426} C_VEL
LIN {X 0,Y 509.884,Z 129.967,A -85,B 0,C 180,E1 -5607.055,E2 -5607.055} C_VEL
LIN {X 0,Y 509.853,Z 129.973,A -85,B 0,C 180,E1 -5609.751,E2 -5609.751} C_VEL
LIN {X 0,Y 509.873,Z 129.969,A -85,B 0,C 180,E1 -5612.775,E2 -5612.775} C_VEL
LIN {X 0,Y 509.836,Z 129.975,A -85,B 0,C 180,E1 -5615.581,E2 -5615.581} C_VEL
LIN {X 0,Y 509.855,Z 129.975,A -85,B 0,C 180,E1 -5618.337,E2 -5618.337} C_VEL
LIN {X 0,Y 509.861,Z 129.971,A -85,B 0,C 180,E1 -5621.424,E2 -5621.424} C_VEL
LIN {X 0,Y 509.852,Z 129.971,A -85,B 0,C 180,E1 -5624.668,E2 -5624.668} C_VEL
LIN {X 0,Y 509.877,Z 129.973,A -85,B 0,C 180,E1 -5628.1,E2 -5628.1} C_VEL
LIN {X 0,Y 509.872,Z 129.968,A -85,B 0,C 180,E1 -5630.65,E2 -5630.65} C_VEL
LIN {X 0,Y 509.826,Z 129.98,A -85,B 0,C 180,E1 -5633.736,E2 -5633.736} C_VEL
LIN {X 0,Y 509.159,Z 130.059,A -85,B 0,C 180,E1 -5634.396,E2 -5634.396} C_VEL
LIN {X 0,Y 506.342,Z 130.413,A -85,B 0,C 180,E1 -5635.468,E2 -5635.468} C_VEL
LIN {X 0,Y 503.95,Z 130.709,A -85,B 0,C 180,E1 -5636.331,E2 -5636.331} C_VEL
LIN {X 0,Y 502.902,Z 130.837,A -85,B 0,C 180,E1 -5636.997,E2 -5636.997} C_VEL
LIN {X 0,Y 502.805,Z 130.849,A -85,B 0,C 180,E1 -5637.223,E2 -5637.223} C_VEL
LIN {X 0,Y 502.81,Z 130.851,A -85,B 0,C 180,E1 -5640.065,E2 -5640.065} C_VEL
LIN {X 0,Y 502.83,Z 130.845,A -85,B 0,C 180,E1 -5642.534,E2 -5642.534} C_VEL
LIN {X 0,Y 502.824,Z 130.852,A -85,B 0,C 180,E1 -5645.299,E2 -5645.299} C_VEL
LIN {X 0,Y 502.789,Z 130.854,A -85,B 0,C 180,E1 -5647.827,E2 -5647.827} C_VEL
LIN {X 0,Y 502.821,Z 130.846,A -85,B 0,C 180,E1 -5650.4,E2 -5650.4} C_VEL
LIN {X 0,Y 502.83,Z 130.848,A -85,B 0,C 180,E1 -5652.932,E2 -5652.932} C_VEL
LIN {X 0,Y 502.847,Z 130.85,A -85,B 0,C 180,E1 -5655.43,E2 -5655.43} C_VEL
LIN {X 0,Y 502.874,Z 130.842,A -85,B 0,C 180,E1 -5658.717,E2 -5658.717} C_VEL
LIN {X 0,Y 502.898,Z 130.837,A -85,B 0,C 180,E1 -5661.967,E2 -5661.967} C_VEL
LIN {X 0,Y 502.939,Z 130.832,A -85,B 0,C 180,E1 -5664.387,E2 -5664.387} C_VEL
LIN {X 0,Y 503.023,Z 130.823,A -85,B 0,C 180,E1 -5667.598,E2 -5667.598} C_VEL
LIN {X 0,Y 503.025,Z 130.821,A -85,B 0,C 180,E1 -5670,E2 -5670} C_VEL
LIN {X 0,Y 503.023,Z 130.823,A -85,B 0,C 180,E1 -5672.403,E2 -5672.403} C_VEL
LIN {X 0,Y 502.939,Z 130.832,A -85,B 0,C 180,E1 -5675.614,E2 -5675.614} C_VEL
LIN {X 0,Y 502.899,Z 130.837,A -85,B 0,C 180,E1 -5678.034,E2 -5678.034} C_VEL
LIN {X 0,Y 502.875,Z 130.842,A -85,B 0,C 180,E1 -5681.284,E2 -5681.284} C_VEL
LIN {X 0,Y 502.849,Z 130.851,A -85,B 0,C 180,E1 -5684.571,E2 -5684.571} C_VEL
LIN {X 0,Y 502.871,Z 130.845,A -85,B 0,C 180,E1 -5687.907,E2 -5687.907} C_VEL
LIN {X 0,Y 502.882,Z 131.061,A -85,B 0,C 180,E1 -5688.658,E2 -5688.658} C_VEL
LIN {X 0,Y 503.52,Z 136.509,A -85,B 0,C 180,E1 -5689.784,E2 -5689.784} C_VEL
LIN {X 0,Y 503.283,Z 148.955,A -85,B 0,C 180,E1 -5692.265,E2 -5692.265} C_VEL
LIN {X 0,Y 505.49,Z 160.297,A -85,B 0,C 180,E1 -5692.505,E2 -5692.505} C_VEL
LIN {X 0,Y 504.813,Z 255.376,A -85,B 0,C 180,E1 -5693.894,E2 -5693.894} C_VEL
LIN {X 0,Y 504.586,Z 269.054,A -85,B 0,C 180,E1 -5694.261,E2 -5694.261} C_VEL
LIN {X 0,Y 504.383,Z 281.618,A -85,B 0,C 180,E1 -5694.766,E2 -5694.766} C_VEL
LIN {X 0,Y 504.167,Z 292.632,A -85,B 0,C 180,E1 -5695.36,E2 -5695.36} C_VEL
LIN {X 0,Y 503.738,Z 304.471,A -85,B 0,C 180,E1 -5696.182,E2 -5696.182} C_VEL
LIN {X 0,Y 503.416,Z 315.316,A -85,B 0,C 180,E1 -5697.133,E2 -5697.133} C_VEL
LIN {X 0,Y 503.08,Z 324.386,A -85,B 0,C 180,E1 -5698.117,E2 -5698.117} C_VEL
LIN {X 0,Y 502.816,Z 333.122,A -85,B 0,C 180,E1 -5699.289,E2 -5699.289} C_VEL
LIN {X 0,Y 502.572,Z 340.208,A -85,B 0,C 180,E1 -5700.46,E2 -5700.46} C_VEL
LIN {X 0,Y 502.404,Z 346.408,A -85,B 0,C 180,E1 -5701.739,E2 -5701.739} C_VEL
LIN {X 0,Y 502.24,Z 351.403,A -85,B 0,C 180,E1 -5703.076,E2 -5703.076} C_VEL
LIN {X 0,Y 502.136,Z 354.899,A -85,B 0,C 180,E1 -5704.334,E2 -5704.334} C_VEL
LIN {X 0,Y 502.031,Z 357.501,A -85,B 0,C 180,E1 -5705.714,E2 -5705.714} C_VEL
LIN {X 0,Y 502.008,Z 358.882,A -85,B 0,C 180,E1 -5707.063,E2 -5707.063} C_VEL
LIN {X 0,Y 502.011,Z 359.154,A -85,B 0,C 180,E1 -5708.374,E2 -5708.374} C_VEL
LIN {X 0,Y 502.022,Z 358.407,A -85,B 0,C 180,E1 -5709.65,E2 -5709.65} C_VEL
LIN {X 0,Y 502.107,Z 356.269,A -85,B 0,C 180,E1 -5711.137,E2 -5711.137} C_VEL
LIN {X 0,Y 502.204,Z 353.837,A -85,B 0,C 180,E1 -5712.201,E2 -5712.201} C_VEL
LIN {X 0,Y 502.267,Z 350.473,A -85,B 0,C 180,E1 -5713.314,E2 -5713.314} C_VEL
LIN {X 0,Y 502.416,Z 344.994,A -85,B 0,C 180,E1 -5714.692,E2 -5714.692} C_VEL
LIN {X 0,Y 502.638,Z 339.21,A -85,B 0,C 180,E1 -5715.833,E2 -5715.833} C_VEL
LIN {X 0,Y 502.845,Z 331.678,A -85,B 0,C 180,E1 -5717.039,E2 -5717.039} C_VEL
LIN {X 0,Y 503.162,Z 322.863,A -85,B 0,C 180,E1 -5718.168,E2 -5718.168} C_VEL
LIN {X 0,Y 503.475,Z 313.655,A -85,B 0,C 180,E1 -5719.132,E2 -5719.132} C_VEL
LIN {X 0,Y 503.728,Z 304.21,A -85,B 0,C 180,E1 -5719.945,E2 -5719.945} C_VEL
LIN {X 0,Y 504.147,Z 293.48,A -85,B 0,C 180,E1 -5720.69,E2 -5720.69} C_VEL
LIN {X 0,Y 504.435,Z 282.74,A -85,B 0,C 180,E1 -5721.281,E2 -5721.281} C_VEL
LIN {X 0,Y 504.614,Z 269.791,A -85,B 0,C 180,E1 -5721.812,E2 -5721.812} C_VEL
LIN {X 0,Y 504.822,Z 257.084,A -85,B 0,C 180,E1 -5722.163,E2 -5722.163} C_VEL
LIN {X 0,Y 505.152,Z 209.206,A -85,B 0,C 180,E1 -5722.883,E2 -5722.883} C_VEL
LIN {X 0,Y 505.375,Z 159.124,A -85,B 0,C 180,E1 -5723.617,E2 -5723.617} C_VEL
LIN {X 0,Y 503.344,Z 149.176,A -85,B 0,C 180,E1 -5723.84,E2 -5723.84} C_VEL
LIN {X 0,Y 503.507,Z 136.466,A -85,B 0,C 180,E1 -5726.302,E2 -5726.302} C_VEL
LIN {X 0,Y 502.879,Z 130.848,A -85,B 0,C 180,E1 -5727.449,E2 -5727.449} C_VEL
LIN {X 0,Y 502.825,Z 130.85,A -85,B 0,C 180,E1 -5730.713,E2 -5730.713} C_VEL
LIN {X 0,Y 502.848,Z 130.852,A -85,B 0,C 180,E1 -5733.444,E2 -5733.444} C_VEL
LIN {X 0,Y 502.79,Z 130.86,A -85,B 0,C 180,E1 -5736.96,E2 -5736.96} C_VEL
LIN {X 0,Y 502.839,Z 130.848,A -85,B 0,C 180,E1 -5739.549,E2 -5739.549} C_VEL
LIN {X 0,Y 502.82,Z 130.848,A -85,B 0,C 180,E1 -5742.092,E2 -5742.092} C_VEL
LIN {X 0,Y 502.843,Z 130.848,A -85,B 0,C 180,E1 -5745.43,E2 -5745.43} C_VEL
LIN {X 0,Y 502.88,Z 130.848,A -85,B 0,C 180,E1 -5748.717,E2 -5748.717} C_VEL
LIN {X 0,Y 502.876,Z 130.844,A -85,B 0,C 180,E1 -5751.967,E2 -5751.967} C_VEL
LIN {X 0,Y 502.902,Z 130.846,A -85,B 0,C 180,E1 -5754.387,E2 -5754.387} C_VEL
LIN {X 0,Y 503.014,Z 130.825,A -85,B 0,C 180,E1 -5757.598,E2 -5757.598} C_VEL
LIN {X 0,Y 503.007,Z 130.826,A -85,B 0,C 180,E1 -5760,E2 -5760} C_VEL
LIN {X 0,Y 503.013,Z 130.825,A -85,B 0,C 180,E1 -5762.403,E2 -5762.403} C_VEL
LIN {X 0,Y 502.896,Z 130.841,A -85,B 0,C 180,E1 -5765.614,E2 -5765.614} C_VEL
LIN {X 0,Y 502.851,Z 130.85,A -85,B 0,C 180,E1 -5768.035,E2 -5768.035} C_VEL
LIN {X 0,Y 502.84,Z 130.843,A -85,B 0,C 180,E1 -5771.284,E2 -5771.284} C_VEL
LIN {X 0,Y 502.798,Z 130.848,A -85,B 0,C 180,E1 -5774.573,E2 -5774.573} C_VEL
LIN {X 0,Y 502.775,Z 130.856,A -85,B 0,C 180,E1 -5777.911,E2 -5777.911} C_VEL
LIN {X 0,Y 502.773,Z 130.852,A -85,B 0,C 180,E1 -5780.517,E2 -5780.517} C_VEL
LIN {X 0,Y 502.782,Z 130.855,A -85,B 0,C 180,E1 -5783.041,E2 -5783.041} C_VEL
LIN {X 0,Y 502.764,Z 130.858,A -85,B 0,C 180,E1 -5785.68,E2 -5785.68} C_VEL
LIN {X 0,Y 502.764,Z 130.853,A -85,B 0,C 180,E1 -5788.378,E2 -5788.378} C_VEL
LIN {X 0,Y 502.775,Z 130.855,A -85,B 0,C 180,E1 -5791.494,E2 -5791.494} C_VEL
LIN {X 0,Y 502.792,Z 130.853,A -85,B 0,C 180,E1 -5794.441,E2 -5794.441} C_VEL
LIN {X 0,Y 502.769,Z 130.857,A -85,B 0,C 180,E1 -5797.176,E2 -5797.176} C_VEL
LIN {X 0,Y 502.776,Z 130.854,A -85,B 0,C 180,E1 -5800.017,E2 -5800.017} C_VEL
LIN {X 0,Y 502.751,Z 130.858,A -85,B 0,C 180,E1 -5803.234,E2 -5803.234} C_VEL
LIN {X 0,Y 502.783,Z 130.854,A -85,B 0,C 180,E1 -5805.66,E2 -5805.66} C_VEL
LIN {X 0,Y 502.781,Z 130.857,A -85,B 0,C 180,E1 -5808.93,E2 -5808.93} C_VEL
LIN {X 0,Y 502.795,Z 130.856,A -85,B 0,C 180,E1 -5812.046,E2 -5812.046} C_VEL
LIN {X 0,Y 502.802,Z 130.851,A -85,B 0,C 180,E1 -5815.034,E2 -5815.034} C_VEL
LIN {X 0,Y 502.788,Z 130.861,A -85,B 0,C 180,E1 -5817.915,E2 -5817.915} C_VEL
LIN {X 0,Y 502.817,Z 130.85,A -85,B 0,C 180,E1 -5820.711,E2 -5820.711} C_VEL
LIN {X 0,Y 502.849,Z 130.85,A -85,B 0,C 180,E1 -5823.443,E2 -5823.443} C_VEL
LIN {X 0,Y 502.851,Z 130.874,A -85,B 0,C 180,E1 -5824.658,E2 -5824.658} C_VEL
LIN {X 0,Y 504.472,Z 139.865,A -85,B 0,C 180,E1 -5826.17,E2 -5826.17} C_VEL
LIN {X 0,Y 504.038,Z 157.766,A -85,B 0,C 180,E1 -5828.982,E2 -5828.982} C_VEL
LIN {X 0,Y 503.538,Z 178.02,A -85,B 0,C 180,E1 -5832.117,E2 -5832.117} C_VEL
LIN {X 0,Y 503.182,Z 191.51,A -85,B 0,C 180,E1 -5834.184,E2 -5834.184} C_VEL
LIN {X 0,Y 505.329,Z 206.34,A -85,B 0,C 180,E1 -5834.474,E2 -5834.474} C_VEL
LIN {X 0,Y 504.752,Z 301.144,A -85,B 0,C 180,E1 -5835.871,E2 -5835.871} C_VEL
LIN {X 0,Y 504.448,Z 314.876,A -85,B 0,C 180,E1 -5836.248,E2 -5836.248} C_VEL
LIN {X 0,Y 504.114,Z 327.245,A -85,B 0,C 180,E1 -5836.752,E2 -5836.752} C_VEL
LIN {X 0,Y 503.78,Z 338.959,A -85,B 0,C 180,E1 -5837.398,E2 -5837.398} C_VEL
LIN {X 0,Y 503.414,Z 350.58,A -85,B 0,C 180,E1 -5838.218,E2 -5838.218} C_VEL
LIN {X 0,Y 503.113,Z 360.913,A -85,B 0,C 180,E1 -5839.129,E2 -5839.129} C_VEL
LIN {X 0,Y 502.767,Z 370.192,A -85,B 0,C 180,E1 -5840.14,E2 -5840.14} C_VEL
LIN {X 0,Y 502.484,Z 379.226,A -85,B 0,C 180,E1 -5841.352,E2 -5841.352} C_VEL
LIN {X 0,Y 502.331,Z 386.507,A -85,B 0,C 180,E1 -5842.564,E2 -5842.564} C_VEL
LIN {X 0,Y 502.217,Z 391.42,A -85,B 0,C 180,E1 -5843.572,E2 -5843.572} C_VEL
LIN {X 0,Y 502.171,Z 396.199,A -85,B 0,C 180,E1 -5844.78,E2 -5844.78} C_VEL
LIN {X 0,Y 502.14,Z 399.852,A -85,B 0,C 180,E1 -5845.987,E2 -5845.987} C_VEL
LIN {X 0,Y 502.137,Z 401.739,A -85,B 0,C 180,E1 -5846.79,E2 -5846.79} C_VEL
LIN {X 0,Y 502.125,Z 403.153,A -85,B 0,C 180,E1 -5847.593,E2 -5847.593} C_VEL
LIN {X 0,Y 502.001,Z 404.78,A -85,B 0,C 180,E1 -5849.197,E2 -5849.197} C_VEL
LIN {X 0,Y 501.997,Z 405.005,A -85,B 0,C 180,E1 -5850,E2 -5850} C_VEL
LIN {X 0,Y 502.037,Z 404.187,A -85,B 0,C 180,E1 -5851.604,E2 -5851.604} C_VEL
LIN {X 0,Y 502.125,Z 403.193,A -85,B 0,C 180,E1 -5852.406,E2 -5852.406} C_VEL
LIN {X 0,Y 502.137,Z 401.79,A -85,B 0,C 180,E1 -5853.209,E2 -5853.209} C_VEL
LIN {X 0,Y 502.101,Z 398.835,A -85,B 0,C 180,E1 -5854.415,E2 -5854.415} C_VEL
LIN {X 0,Y 502.191,Z 394.838,A -85,B 0,C 180,E1 -5855.621,E2 -5855.621} C_VEL
LIN {X 0,Y 502.291,Z 388.782,A -85,B 0,C 180,E1 -5857.012,E2 -5857.012} C_VEL
LIN {X 0,Y 502.445,Z 381.955,A -85,B 0,C 180,E1 -5858.243,E2 -5858.243} C_VEL
LIN {X 0,Y 502.672,Z 373.612,A -85,B 0,C 180,E1 -5859.455,E2 -5859.455} C_VEL
LIN {X 0,Y 502.949,Z 365.046,A -85,B 0,C 180,E1 -5860.466,E2 -5860.466} C_VEL
LIN {X 0,Y 503.333,Z 354.469,A -85,B 0,C 180,E1 -5861.476,E2 -5861.476} C_VEL
LIN {X 0,Y 503.635,Z 342.968,A -85,B 0,C 180,E1 -5862.36,E2 -5862.36} C_VEL
LIN {X 0,Y 503.974,Z 332.492,A -85,B 0,C 180,E1 -5862.995,E2 -5862.995} C_VEL
LIN {X 0,Y 504.304,Z 320.591,A -85,B 0,C 180,E1 -5863.55,E2 -5863.55} C_VEL
LIN {X 0,Y 504.619,Z 306.865,A -85,B 0,C 180,E1 -5864.003,E2 -5864.003} C_VEL
LIN {X 0,Y 504.852,Z 294.486,A -85,B 0,C 180,E1 -5864.254,E2 -5864.254} C_VEL
LIN {X 0,Y 505.223,Z 205.65,A -85,B 0,C 180,E1 -5865.542,E2 -5865.542} C_VEL
LIN {X 0,Y 503.214,Z 191.919,A -85,B 0,C 180,E1 -5865.816,E2 -5865.816} C_VEL
LIN {X 0,Y 503.765,Z 171.857,A -85,B 0,C 180,E1 -5868.926,E2 -5868.926} C_VEL
LIN {X 0,Y 504.357,Z 151.667,A -85,B 0,C 180,E1 -5872.1,E2 -5872.1} C_VEL
LIN {X 0,Y 504.688,Z 140.878,A -85,B 0,C 180,E1 -5873.818,E2 -5873.818} C_VEL
LIN {X 0,Y 502.859,Z 130.849,A -85,B 0,C 180,E1 -5875.564,E2 -5875.564} C_VEL
LIN {X 0,Y 502.838,Z 130.852,A -85,B 0,C 180,E1 -5878.372,E2 -5878.372} C_VEL
LIN {X 0,Y 502.794,Z 130.852,A -85,B 0,C 180,E1 -5881.498,E2 -5881.498} C_VEL
LIN {X 0,Y 502.805,Z 130.858,A -85,B 0,C 180,E1 -5883.993,E2 -5883.993} C_VEL
LIN {X 0,Y 502.778,Z 130.852,A -85,B 0,C 180,E1 -5887.177,E2 -5887.177} C_VEL
LIN {X 0,Y 502.788,Z 130.857,A -85,B 0,C 180,E1 -5890.015,E2 -5890.015} C_VEL
LIN {X 0,Y 502.803,Z 130.852,A -85,B 0,C 180,E1 -5892.199,E2 -5892.199} C_VEL
LIN {X 0,Y 502.786,Z 130.855,A -85,B 0,C 180,E1 -5895.469,E2 -5895.469} C_VEL
LIN {X 0,Y 502.82,Z 130.847,A -85,B 0,C 180,E1 -5898.934,E2 -5898.934} C_VEL
LIN {X 0,Y 502.793,Z 130.853,A -85,B 0,C 180,E1 -5902.046,E2 -5902.046} C_VEL
LIN {X 0,Y 502.795,Z 130.852,A -85,B 0,C 180,E1 -5905.033,E2 -5905.033} C_VEL
LIN {X 0,Y 502.781,Z 130.855,A -85,B 0,C 180,E1 -5907.915,E2 -5907.915} C_VEL
LIN {X 0,Y 502.822,Z 130.847,A -85,B 0,C 180,E1 -5910.712,E2 -5910.712} C_VEL
LIN {X 0,Y 502.862,Z 130.85,A -85,B 0,C 180,E1 -5913.439,E2 -5913.439} C_VEL
LIN {X 0,Y 502.784,Z 130.852,A -85,B 0,C 180,E1 -5916.085,E2 -5916.085} C_VEL
LIN {X 0,Y 502.782,Z 130.853,A -85,B 0,C 180,E1 -5918.688,E2 -5918.688} C_VEL
LIN {X 0,Y 502.825,Z 130.855,A -85,B 0,C 180,E1 -5921.248,E2 -5921.248} C_VEL
LIN {X 0,Y 502.847,Z 130.845,A -85,B 0,C 180,E1 -5924.6,E2 -5924.6} C_VEL
LIN {X 0,Y 502.875,Z 130.84,A -85,B 0,C 180,E1 -5928.039,E2 -5928.039} C_VEL
LIN {X 0,Y 502.872,Z 130.847,A -85,B 0,C 180,E1 -5931.156,E2 -5931.156} C_VEL
LIN {X 0,Y 502.906,Z 130.837,A -85,B 0,C 180,E1 -5933.581,E2 -5933.581} C_VEL
LIN {X 0,Y 502.897,Z 130.844,A -85,B 0,C 180,E1 -5936.795,E2 -5936.795} C_VEL
LIN {X 0,Y 503.032,Z 130.824,A -85,B 0,C 180,E1 -5939.199,E2 -5939.199} C_VEL
LIN {X 0,Y 502.898,Z 130.837,A -85,B 0,C 180,E1 -5941.601,E2 -5941.601} C_VEL
LIN {X 0,Y 502.895,Z 130.84,A -85,B 0,C 180,E1 -5943.204,E2 -5943.204} C_VEL
LIN {X 0,Y 502.905,Z 130.841,A -85,B 0,C 180,E1 -5946.419,E2 -5946.419} C_VEL
LIN {X 0,Y 502.872,Z 130.846,A -85,B 0,C 180,E1 -5948.843,E2 -5948.843} C_VEL
LIN {X 0,Y 502.843,Z 130.846,A -85,B 0,C 180,E1 -5952.101,E2 -5952.101} C_VEL
LIN {X 0,Y 502.846,Z 130.844,A -85,B 0,C 180,E1 -5955.399,E2 -5955.399} C_VEL
LIN {X 0,Y 502.843,Z 130.848,A -85,B 0,C 180,E1 -5958.122,E2 -5958.122} C_VEL
LIN {X 0,Y 502.825,Z 130.853,A -85,B 0,C 180,E1 -5960.536,E2 -5960.536} C_VEL
LIN {X 0,Y 502.788,Z 130.852,A -85,B 0,C 180,E1 -5963.04,E2 -5963.04} C_VEL
LIN {X 0,Y 502.838,Z 130.846,A -85,B 0,C 180,E1 -5965.675,E2 -5965.675} C_VEL
LIN {X 0,Y 502.837,Z 130.852,A -85,B 0,C 180,E1 -5968.372,E2 -5968.372} C_VEL
LIN {X 0,Y 502.792,Z 130.851,A -85,B 0,C 180,E1 -5971.499,E2 -5971.499} C_VEL
LIN {X 0,Y 502.801,Z 130.853,A -85,B 0,C 180,E1 -5974.444,E2 -5974.444} C_VEL
LIN {X 0,Y 502.777,Z 130.852,A -85,B 0,C 180,E1 -5977.178,E2 -5977.178} C_VEL
LIN {X 0,Y 502.822,Z 130.855,A -85,B 0,C 180,E1 -5980.011,E2 -5980.011} C_VEL
LIN {X 0,Y 502.818,Z 130.852,A -85,B 0,C 180,E1 -5982.202,E2 -5982.202} C_VEL
LIN {X 0,Y 502.796,Z 130.852,A -85,B 0,C 180,E1 -5985.468,E2 -5985.468} C_VEL
LIN {X 0,Y 502.83,Z 130.854,A -85,B 0,C 180,E1 -5987.865,E2 -5987.865} C_VEL
LIN {X 0,Y 502.817,Z 130.847,A -85,B 0,C 180,E1 -5991.026,E2 -5991.026} C_VEL
LIN {X 0,Y 502.779,Z 130.855,A -85,B 0,C 180,E1 -5994.168,E2 -5994.168} C_VEL
LIN {X 0,Y 502.805,Z 130.849,A -85,B 0,C 180,E1 -5997.223,E2 -5997.223} C_VEL
LIN {X 0,Y 502.104,Z 130.942,A -85,B 0,C 180,E1 -5997.892,E2 -5997.892} C_VEL
LIN {X 0,Y 499.239,Z 131.294,A -85,B 0,C 180,E1 -5998.978,E2 -5998.978} C_VEL
LIN {X 0,Y 496.843,Z 131.596,A -85,B 0,C 180,E1 -5999.852,E2 -5999.852} C_VEL
LIN {X 0,Y 495.826,Z 131.718,A -85,B 0,C 180,E1 -6000.528,E2 -6000.528} C_VEL
LIN {X 0,Y 495.748,Z 131.728,A -85,B 0,C 180,E1 -6000.757,E2 -6000.757} C_VEL
LIN {X 0,Y 495.794,Z 131.725,A -85,B 0,C 180,E1 -6003.933,E2 -6003.933} C_VEL
LIN {X 0,Y 495.753,Z 131.731,A -85,B 0,C 180,E1 -6007.14,E2 -6007.14} C_VEL
LIN {X 0,Y 495.773,Z 131.725,A -85,B 0,C 180,E1 -6010.11,E2 -6010.11} C_VEL
LIN {X 0,Y 495.782,Z 131.724,A -85,B 0,C 180,E1 -6012.682,E2 -6012.682} C_VEL
LIN {X 0,Y 495.79,Z 131.73,A -85,B 0,C 180,E1 -6015.218,E2 -6015.218} C_VEL
LIN {X 0,Y 495.848,Z 131.716,A -85,B 0,C 180,E1 -6018.555,E2 -6018.555} C_VEL
LIN {X 0,Y 495.87,Z 131.713,A -85,B 0,C 180,E1 -6021.852,E2 -6021.852} C_VEL
LIN {X 0,Y 495.896,Z 131.709,A -85,B 0,C 180,E1 -6024.307,E2 -6024.307} C_VEL
LIN {X 0,Y 495.991,Z 131.699,A -85,B 0,C 180,E1 -6027.564,E2 -6027.564} C_VEL
LIN {X 0,Y 495.996,Z 131.697,A -85,B 0,C 180,E1 -6030,E2 -6030} C_VEL
LIN {X 0,Y 495.992,Z 131.699,A -85,B 0,C 180,E1 -6032.437,E2 -6032.437} C_VEL
LIN {X 0,Y 495.897,Z 131.709,A -85,B 0,C 180,E1 -6035.694,E2 -6035.694} C_VEL
LIN {X 0,Y 495.871,Z 131.713,A -85,B 0,C 180,E1 -6038.148,E2 -6038.148} C_VEL
LIN {X 0,Y 495.849,Z 131.716,A -85,B 0,C 180,E1 -6041.446,E2 -6041.446} C_VEL
LIN {X 0,Y 495.792,Z 131.731,A -85,B 0,C 180,E1 -6044.783,E2 -6044.783} C_VEL
LIN {X 0,Y 495.83,Z 131.726,A -85,B 0,C 180,E1 -6048.257,E2 -6048.257} C_VEL
LIN {X 0,Y 495.831,Z 131.866,A -85,B 0,C 180,E1 -6048.507,E2 -6048.507} C_VEL
LIN {X 0,Y 496.555,Z 137.287,A -85,B 0,C 180,E1 -6049.643,E2 -6049.643} C_VEL
LIN {X 0,Y 496.355,Z 149.194,A -85,B 0,C 180,E1 -6052.038,E2 -6052.038} C_VEL
LIN {X 0,Y 498.687,Z 162.029,A -85,B 0,C 180,E1 -6052.311,E2 -6052.311} C_VEL
LIN {X 0,Y 497.946,Z 256.39,A -85,B 0,C 180,E1 -6053.716,E2 -6053.716} C_VEL
LIN {X 0,Y 497.7,Z 269.469,A -85,B 0,C 180,E1 -6054.075,E2 -6054.075} C_VEL
LIN {X 0,Y 497.5,Z 281.705,A -85,B 0,C 180,E1 -6054.574,E2 -6054.574} C_VEL
LIN {X 0,Y 497.226,Z 293.653,A -85,B 0,C 180,E1 -6055.232,E2 -6055.232} C_VEL
LIN {X 0,Y 496.799,Z 304.685,A -85,B 0,C 180,E1 -6056.012,E2 -6056.012} C_VEL
LIN {X 0,Y 496.44,Z 315.165,A -85,B 0,C 180,E1 -6056.938,E2 -6056.938} C_VEL
LIN {X 0,Y 496.118,Z 323.787,A -85,B 0,C 180,E1 -6057.871,E2 -6057.871} C_VEL
LIN {X 0,Y 495.813,Z 332.623,A -85,B 0,C 180,E1 -6059.045,E2 -6059.045} C_VEL
LIN {X 0,Y 495.534,Z 340.615,A -85,B 0,C 180,E1 -6060.372,E2 -6060.372} C_VEL
LIN {X 0,Y 495.346,Z 346.786,A -85,B 0,C 180,E1 -6061.666,E2 -6061.666} C_VEL
LIN {X 0,Y 495.152,Z 352.098,A -85,B 0,C 180,E1 -6063.132,E2 -6063.132} C_VEL
LIN {X 0,Y 495.013,Z 355.923,A -85,B 0,C 180,E1 -6064.605,E2 -6064.605} C_VEL
LIN {X 0,Y 494.933,Z 358.211,A -85,B 0,C 180,E1 -6065.964,E2 -6065.964} C_VEL
LIN {X 0,Y 494.917,Z 359.369,A -85,B 0,C 180,E1 -6067.325,E2 -6067.325} C_VEL
LIN {X 0,Y 494.929,Z 359.423,A -85,B 0,C 180,E1 -6068.668,E2 -6068.668} C_VEL
LIN {X 0,Y 494.952,Z 358.477,A -85,B 0,C 180,E1 -6069.937,E2 -6069.937} C_VEL
LIN {X 0,Y 495.032,Z 356.566,A -85,B 0,C 180,E1 -6071.198,E2 -6071.198} C_VEL
LIN {X 0,Y 495.127,Z 353.725,A -85,B 0,C 180,E1 -6072.431,E2 -6072.431} C_VEL
LIN {X 0,Y 495.219,Z 349.955,A -85,B 0,C 180,E1 -6073.634,E2 -6073.634} C_VEL
LIN {X 0,Y 495.376,Z 345.18,A -85,B 0,C 180,E1 -6074.818,E2 -6074.818} C_VEL
LIN {X 0,Y 495.616,Z 339.301,A -85,B 0,C 180,E1 -6075.987,E2 -6075.987} C_VEL
LIN {X 0,Y 495.828,Z 332.254,A -85,B 0,C 180,E1 -6077.129,E2 -6077.129} C_VEL
LIN {X 0,Y 496.149,Z 323.632,A -85,B 0,C 180,E1 -6078.26,E2 -6078.26} C_VEL
LIN {X 0,Y 496.538,Z 313.06,A -85,B 0,C 180,E1 -6079.377,E2 -6079.377} C_VEL
LIN {X 0,Y 496.87,Z 301.975,A -85,B 0,C 180,E1 -6080.31,E2 -6080.31} C_VEL
LIN {X 0,Y 497.333,Z 290.068,A -85,B 0,C 180,E1 -6081.091,E2 -6081.091} C_VEL
LIN {X 0,Y 497.696,Z 277.493,A -85,B 0,C 180,E1 -6081.721,E2 -6081.721} C_VEL
LIN {X 0,Y 497.82,Z 265.409,A -85,B 0,C 180,E1 -6082.157,E2 -6082.157} C_VEL
LIN {X 0,Y 498.031,Z 252.501,A -85,B 0,C 180,E1 -6082.454,E2 -6082.454} C_VEL
LIN {X 0,Y 498.62,Z 160.402,A -85,B 0,C 180,E1 -6083.822,E2 -6083.822} C_VEL
LIN {X 0,Y 496.402,Z 149.489,A -85,B 0,C 180,E1 -6084.072,E2 -6084.072} C_VEL
LIN {X 0,Y 496.527,Z 137.083,A -85,B 0,C 180,E1 -6086.495,E2 -6086.495} C_VEL
LIN {X 0,Y 495.808,Z 131.729,A -85,B 0,C 180,E1 -6087.587,E2 -6087.587} C_VEL
LIN {X 0,Y 495.768,Z 131.728,A -85,B 0,C 180,E1 -6090.254,E2 -6090.254} C_VEL
LIN {X 0,Y 495.809,Z 131.73,A -85,B 0,C 180,E1 -6093.256,E2 -6093.256} C_VEL
LIN {X 0,Y 495.743,Z 131.734,A -85,B 0,C 180,E1 -6096.613,E2 -6096.613} C_VEL
LIN {X 0,Y 495.782,Z 131.73,A -85,B 0,C 180,E1 -6099.325,E2 -6099.325} C_VEL
LIN {X 0,Y 495.782,Z 131.725,A -85,B 0,C 180,E1 -6101.829,E2 -6101.829} C_VEL
LIN {X 0,Y 495.828,Z 131.724,A -85,B 0,C 180,E1 -6104.549,E2 -6104.549} C_VEL
LIN {X 0,Y 495.833,Z 131.721,A -85,B 0,C 180,E1 -6107.966,E2 -6107.966} C_VEL
LIN {X 0,Y 495.836,Z 131.722,A -85,B 0,C 180,E1 -6111.031,E2 -6111.031} C_VEL
LIN {X 0,Y 495.829,Z 131.72,A -85,B 0,C 180,E1 -6113.489,E2 -6113.489} C_VEL
LIN {X 0,Y 495.715,Z 131.735,A -85,B 0,C 180,E1 -6115.935,E2 -6115.935} C_VEL
LIN {X 0,Y 495.981,Z 131.701,A -85,B 0,C 180,E1 -6117.564,E2 -6117.564} C_VEL
LIN {X 0,Y 495.976,Z 131.702,A -85,B 0,C 180,E1 -6120,E2 -6120} C_VEL
LIN {X 0,Y 495.979,Z 131.701,A -85,B 0,C 180,E1 -6122.437,E2 -6122.437} C_VEL
LIN {X 0,Y 495.854,Z 131.719,A -85,B 0,C 180,E1 -6125.694,E2 -6125.694} C_VEL
LIN {X 0,Y 495.815,Z 131.725,A -85,B 0,C 180,E1 -6128.149,E2 -6128.149} C_VEL
LIN {X 0,Y 495.818,Z 131.719,A -85,B 0,C 180,E1 -6131.446,E2 -6131.446} C_VEL
LIN {X 0,Y 495.747,Z 131.726,A -85,B 0,C 180,E1 -6134.785,E2 -6134.785} C_VEL
LIN {X 0,Y 495.739,Z 131.729,A -85,B 0,C 180,E1 -6138.174,E2 -6138.174} C_VEL
LIN {X 0,Y 495.726,Z 131.737,A -85,B 0,C 180,E1 -6141.63,E2 -6141.63} C_VEL
LIN {X 0,Y 495.701,Z 131.733,A -85,B 0,C 180,E1 -6144.278,E2 -6144.278} C_VEL
LIN {X 0,Y 495.722,Z 131.736,A -85,B 0,C 180,E1 -6146.98,E2 -6146.98} C_VEL
LIN {X 0,Y 495.7,Z 131.736,A -85,B 0,C 180,E1 -6149.751,E2 -6149.751} C_VEL
LIN {X 0,Y 495.753,Z 131.729,A -85,B 0,C 180,E1 -6152.596,E2 -6152.596} C_VEL
LIN {X 0,Y 495.748,Z 131.73,A -85,B 0,C 180,E1 -6155.538,E2 -6155.538} C_VEL
LIN {X 0,Y 495.762,Z 131.732,A -85,B 0,C 180,E1 -6158.767,E2 -6158.767} C_VEL
LIN {X 0,Y 495.728,Z 131.731,A -85,B 0,C 180,E1 -6161.784,E2 -6161.784} C_VEL
LIN {X 0,Y 495.742,Z 131.733,A -85,B 0,C 180,E1 -6165.141,E2 -6165.141} C_VEL
LIN {X 0,Y 495.749,Z 131.735,A -85,B 0,C 180,E1 -6168.217,E2 -6168.217} C_VEL
LIN {X 0,Y 495.75,Z 131.73,A -85,B 0,C 180,E1 -6171.408,E2 -6171.408} C_VEL
LIN {X 0,Y 495.75,Z 131.735,A -85,B 0,C 180,E1 -6174.462,E2 -6174.462} C_VEL
LIN {X 0,Y 495.772,Z 131.73,A -85,B 0,C 180,E1 -6177.405,E2 -6177.405} C_VEL
LIN {X 0,Y 495.767,Z 131.734,A -85,B 0,C 180,E1 -6180.253,E2 -6180.253} C_VEL
LIN {X 0,Y 495.779,Z 131.729,A -85,B 0,C 180,E1 -6183.262,E2 -6183.262} C_VEL
LIN {X 0,Y 495.835,Z 131.912,A -85,B 0,C 180,E1 -6184.498,E2 -6184.498} C_VEL
LIN {X 0,Y 497.493,Z 140.891,A -85,B 0,C 180,E1 -6186.037,E2 -6186.037} C_VEL
LIN {X 0,Y 497.276,Z 151.826,A -85,B 0,C 180,E1 -6187.786,E2 -6187.786} C_VEL
LIN {X 0,Y 496.751,Z 170.89,A -85,B 0,C 180,E1 -6190.795,E2 -6190.795} C_VEL
LIN {X 0,Y 496.163,Z 191.157,A -85,B 0,C 180,E1 -6193.952,E2 -6193.952} C_VEL
LIN {X 0,Y 498.485,Z 208.283,A -85,B 0,C 180,E1 -6194.288,E2 -6194.288} C_VEL
LIN {X 0,Y 497.888,Z 300.719,A -85,B 0,C 180,E1 -6195.672,E2 -6195.672} C_VEL
LIN {X 0,Y 497.557,Z 313.704,A -85,B 0,C 180,E1 -6196.027,E2 -6196.027} C_VEL
LIN {X 0,Y 497.242,Z 325.751,A -85,B 0,C 180,E1 -6196.513,E2 -6196.513} C_VEL
LIN {X 0,Y 496.874,Z 337.347,A -85,B 0,C 180,E1 -6197.14,E2 -6197.14} C_VEL
LIN {X 0,Y 496.428,Z 348.896,A -85,B 0,C 180,E1 -6197.946,E2 -6197.946} C_VEL
LIN {X 0,Y 496.067,Z 359.47,A -85,B 0,C 180,E1 -6198.87,E2 -6198.87} C_VEL
LIN {X 0,Y 495.763,Z 368.118,A -85,B 0,C 180,E1 -6199.793,E2 -6199.793} C_VEL
LIN {X 0,Y 495.528,Z 376.099,A -85,B 0,C 180,E1 -6200.818,E2 -6200.818} C_VEL
LIN {X 0,Y 495.31,Z 383.898,A -85,B 0,C 180,E1 -6202.047,E2 -6202.047} C_VEL
LIN {X 0,Y 495.18,Z 389.236,A -85,B 0,C 180,E1 -6203.071,E2 -6203.071} C_VEL
LIN {X 0,Y 495.105,Z 394.415,A -85,B 0,C 180,E1 -6204.297,E2 -6204.297} C_VEL
LIN {X 0,Y 495.007,Z 398.433,A -85,B 0,C 180,E1 -6205.521,E2 -6205.521} C_VEL
LIN {X 0,Y 495.057,Z 401.409,A -85,B 0,C 180,E1 -6206.744,E2 -6206.744} C_VEL
LIN {X 0,Y 495.029,Z 402.826,A -85,B 0,C 180,E1 -6207.558,E2 -6207.558} C_VEL
LIN {X 0,Y 494.92,Z 404.456,A -85,B 0,C 180,E1 -6209.186,E2 -6209.186} C_VEL
LIN {X 0,Y 494.914,Z 404.682,A -85,B 0,C 180,E1 -6210,E2 -6210} C_VEL
LIN {X 0,Y 494.964,Z 403.866,A -85,B 0,C 180,E1 -6211.627,E2 -6211.627} C_VEL
LIN {X 0,Y 495.029,Z 402.871,A -85,B 0,C 180,E1 -6212.441,E2 -6212.441} C_VEL
LIN {X 0,Y 495.057,Z 401.467,A -85,B 0,C 180,E1 -6213.255,E2 -6213.255} C_VEL
LIN {X 0,Y 495.006,Z 398.51,A -85,B 0,C 180,E1 -6214.478,E2 -6214.478} C_VEL
LIN {X 0,Y 495.105,Z 394.51,A -85,B 0,C 180,E1 -6215.702,E2 -6215.702} C_VEL
LIN {X 0,Y 495.239,Z 388.347,A -85,B 0,C 180,E1 -6217.132,E2 -6217.132} C_VEL
LIN {X 0,Y 495.371,Z 381.615,A -85,B 0,C 180,E1 -6218.361,E2 -6218.361} C_VEL
LIN {X 0,Y 495.632,Z 373.266,A -85,B 0,C 180,E1 -6219.591,E2 -6219.591} C_VEL
LIN {X 0,Y 495.952,Z 364.688,A -85,B 0,C 180,E1 -6220.615,E2 -6220.615} C_VEL
LIN {X 0,Y 496.322,Z 354.098,A -85,B 0,C 180,E1 -6221.641,E2 -6221.641} C_VEL
LIN {X 0,Y 496.625,Z 343.695,A -85,B 0,C 180,E1 -6222.457,E2 -6222.457} C_VEL
LIN {X 0,Y 497.017,Z 332.088,A -85,B 0,C 180,E1 -6223.18,E2 -6223.18} C_VEL
LIN {X 0,Y 497.417,Z 318.855,A -85,B 0,C 180,E1 -6223.793,E2 -6223.793} C_VEL
LIN {X 0,Y 497.77,Z 305.465,A -85,B 0,C 180,E1 -6224.226,E2 -6224.226} C_VEL
LIN {X 0,Y 497.977,Z 290.32,A -85,B 0,C 180,E1 -6224.507,E2 -6224.507} C_VEL
LIN {X 0,Y 498.362,Z 206.349,A -85,B 0,C 180,E1 -6225.745,E2 -6225.745} C_VEL
LIN {X 0,Y 496.221,Z 191.665,A -85,B 0,C 180,E1 -6226.036,E2 -6226.036} C_VEL
LIN {X 0,Y 496.811,Z 171.547,A -85,B 0,C 180,E1 -6229.202,E2 -6229.202} C_VEL
LIN {X 0,Y 497.495,Z 150.008,A -85,B 0,C 180,E1 -6232.64,E2 -6232.64} C_VEL
LIN {X 0,Y 497.725,Z 141.921,A -85,B 0,C 180,E1 -6233.95,E2 -6233.95} C_VEL
LIN {X 0,Y 495.817,Z 131.726,A -85,B 0,C 180,E1 -6235.727,E2 -6235.727} C_VEL
LIN {X 0,Y 495.77,Z 131.729,A -85,B 0,C 180,E1 -6238.814,E2 -6238.814} C_VEL
LIN {X 0,Y 495.756,Z 131.731,A -85,B 0,C 180,E1 -6241.725,E2 -6241.725} C_VEL
LIN {X 0,Y 495.769,Z 131.726,A -85,B 0,C 180,E1 -6244.693,E2 -6244.693} C_VEL
LIN {X 0,Y 495.73,Z 131.734,A -85,B 0,C 180,E1 -6247.561,E2 -6247.561} C_VEL
LIN {X 0,Y 495.766,Z 131.725,A -85,B 0,C 180,E1 -6250.699,E2 -6250.699} C_VEL
LIN {X 0,Y 495.727,Z 131.736,A -85,B 0,C 180,E1 -6254.001,E2 -6254.001} C_VEL
LIN {X 0,Y 495.726,Z 131.732,A -85,B 0,C 180,E1 -6257.116,E2 -6257.116} C_VEL
LIN {X 0,Y 495.758,Z 131.731,A -85,B 0,C 180,E1 -6259.952,E2 -6259.952} C_VEL
LIN {X 0,Y 495.727,Z 131.73,A -85,B 0,C 180,E1 -6262.553,E2 -6262.553} C_VEL
LIN {X 0,Y 495.77,Z 131.732,A -85,B 0,C 180,E1 -6265.456,E2 -6265.456} C_VEL
LIN {X 0,Y 495.753,Z 131.727,A -85,B 0,C 180,E1 -6268.363,E2 -6268.363} C_VEL
LIN {X 0,Y 495.786,Z 131.73,A -85,B 0,C 180,E1 -6271.507,E2 -6271.507} C_VEL
LIN {X 0,Y 495.79,Z 131.724,A -85,B 0,C 180,E1 -6273.932,E2 -6273.932} C_VEL
LIN {X 0,Y 495.759,Z 131.732,A -85,B 0,C 180,E1 -6277.139,E2 -6277.139} C_VEL
LIN {X 0,Y 495.769,Z 131.725,A -85,B 0,C 180,E1 -6280.109,E2 -6280.109} C_VEL
LIN {X 0,Y 495.763,Z 131.728,A -85,B 0,C 180,E1 -6282.68,E2 -6282.68} C_VEL
LIN {X 0,Y 495.789,Z 131.73,A -85,B 0,C 180,E1 -6285.217,E2 -6285.217} C_VEL
LIN {X 0,Y 495.85,Z 131.717,A -85,B 0,C 180,E1 -6288.554,E2 -6288.554} C_VEL
LIN {X 0,Y 495.872,Z 131.712,A -85,B 0,C 180,E1 -6291.852,E2 -6291.852} C_VEL
LIN {X 0,Y 495.889,Z 131.711,A -85,B 0,C 180,E1 -6294.306,E2 -6294.306} C_VEL
LIN {X 0,Y 495.993,Z 131.698,A -85,B 0,C 180,E1 -6297.563,E2 -6297.563} C_VEL
LIN {X 0,Y 495.997,Z 131.697,A -85,B 0,C 180,E1 -6300,E2 -6300} C_VEL
LIN {X 0,Y 495.993,Z 131.701,A -85,B 0,C 180,E1 -6302.436,E2 -6302.436} C_VEL
LIN {X 0,Y 495.889,Z 131.71,A -85,B 0,C 180,E1 -6305.693,E2 -6305.693} C_VEL
LIN {X 0,Y 495.871,Z 131.714,A -85,B 0,C 180,E1 -6308.148,E2 -6308.148} C_VEL
LIN {X 0,Y 495.849,Z 131.715,A -85,B 0,C 180,E1 -6311.445,E2 -6311.445} C_VEL
LIN {X 0,Y 495.792,Z 131.727,A -85,B 0,C 180,E1 -6314.782,E2 -6314.782} C_VEL
LIN {X 0,Y 495.784,Z 131.723,A -85,B 0,C 180,E1 -6317.318,E2 -6317.318} C_VEL
LIN {X 0,Y 495.774,Z 131.726,A -85,B 0,C 180,E1 -6319.89,E2 -6319.89} C_VEL
LIN {X 0,Y 495.756,Z 131.729,A -85,B 0,C 180,E1 -6322.861,E2 -6322.861} C_VEL
LIN {X 0,Y 495.796,Z 131.727,A -85,B 0,C 180,E1 -6326.067,E2 -6326.067} C_VEL
LIN {X 0,Y 495.768,Z 131.727,A -85,B 0,C 180,E1 -6328.814,E2 -6328.814} C_VEL
LIN {X 0,Y 495.755,Z 131.729,A -85,B 0,C 180,E1 -6331.726,E2 -6331.726} C_VEL
LIN {X 0,Y 495.771,Z 131.726,A -85,B 0,C 180,E1 -6334.695,E2 -6334.695} C_VEL
LIN {X 0,Y 495.728,Z 131.732,A -85,B 0,C 180,E1 -6337.561,E2 -6337.561} C_VEL
LIN {X 0,Y 495.789,Z 131.731,A -85,B 0,C 180,E1 -6340.052,E2 -6340.052} C_VEL
LIN {X 0,Y 495.758,Z 131.726,A -85,B 0,C 180,E1 -6342.879,E2 -6342.879} C_VEL
LIN {X 0,Y 495.732,Z 131.737,A -85,B 0,C 180,E1 -6345.999,E2 -6345.999} C_VEL
LIN {X 0,Y 495.764,Z 131.726,A -85,B 0,C 180,E1 -6348.705,E2 -6348.705} C_VEL
LIN {X 0,Y 495.759,Z 131.73,A -85,B 0,C 180,E1 -6351.41,E2 -6351.41} C_VEL
LIN {X 0,Y 495.751,Z 131.728,A -85,B 0,C 180,E1 -6354.463,E2 -6354.463} C_VEL
LIN {X 0,Y 495.764,Z 131.73,A -85,B 0,C 180,E1 -6357.406,E2 -6357.406} C_VEL
LIN {X 0,Y 495.761,Z 131.727,A -85,B 0,C 180,E1 -6360.254,E2 -6360.254} C_VEL
LIN {X 0,Y 495.748,Z 131.728,A -85,B 0,C 180,E1 -6360.757,E2 -6360.757} C_VEL
LIN {X 0,Y 495.092,Z 131.816,A -85,B 0,C 180,E1 -6361.436,E2 -6361.436} C_VEL
LIN {X 0,Y 492.24,Z 132.168,A -85,B 0,C 180,E1 -6362.539,E2 -6362.539} C_VEL
LIN {X 0,Y 489.833,Z 132.471,A -85,B 0,C 180,E1 -6363.427,E2 -6363.427} C_VEL
LIN {X 0,Y 488.816,Z 132.593,A -85,B 0,C 180,E1 -6364.114,E2 -6364.114} C_VEL
LIN {X 0,Y 488.742,Z 132.601,A -85,B 0,C 180,E1 -6364.346,E2 -6364.346} C_VEL
LIN {X 0,Y 488.716,Z 132.608,A -85,B 0,C 180,E1 -6367.153,E2 -6367.153} C_VEL
LIN {X 0,Y 488.724,Z 132.606,A -85,B 0,C 180,E1 -6369.811,E2 -6369.811} C_VEL
LIN {X 0,Y 488.73,Z 132.602,A -85,B 0,C 180,E1 -6372.424,E2 -6372.424} C_VEL
LIN {X 0,Y 488.76,Z 132.602,A -85,B 0,C 180,E1 -6375,E2 -6375} C_VEL
LIN {X 0,Y 488.802,Z 132.593,A -85,B 0,C 180,E1 -6378.388,E2 -6378.388} C_VEL
LIN {X 0,Y 488.814,Z 132.593,A -85,B 0,C 180,E1 -6381.734,E2 -6381.734} C_VEL
LIN {X 0,Y 488.856,Z 132.586,A -85,B 0,C 180,E1 -6384.225,E2 -6384.225} C_VEL
LIN {X 0,Y 488.959,Z 132.576,A -85,B 0,C 180,E1 -6387.529,E2 -6387.529} C_VEL
LIN {X 0,Y 488.951,Z 132.581,A -85,B 0,C 180,E1 -6390.824,E2 -6390.824} C_VEL
LIN {X 0,Y 488.959,Z 132.576,A -85,B 0,C 180,E1 -6392.472,E2 -6392.472} C_VEL
LIN {X 0,Y 488.856,Z 132.586,A -85,B 0,C 180,E1 -6395.776,E2 -6395.776} C_VEL
LIN {X 0,Y 488.815,Z 132.593,A -85,B 0,C 180,E1 -6398.267,E2 -6398.267} C_VEL
LIN {X 0,Y 488.803,Z 132.593,A -85,B 0,C 180,E1 -6401.613,E2 -6401.613} C_VEL
LIN {X 0,Y 488.763,Z 132.604,A -85,B 0,C 180,E1 -6405.001,E2 -6405.001} C_VEL
LIN {X 0,Y 488.794,Z 132.628,A -85,B 0,C 180,E1 -6408.341,E2 -6408.341} C_VEL
LIN {X 0,Y 489.572,Z 139.163,A -85,B 0,C 180,E1 -6409.716,E2 -6409.716} C_VEL
LIN {X 0,Y 489.366,Z 149.447,A -85,B 0,C 180,E1 -6411.804,E2 -6411.804} C_VEL
LIN {X 0,Y 491.837,Z 162.002,A -85,B 0,C 180,E1 -6412.086,E2 -6412.086} C_VEL
LIN {X 0,Y 491.091,Z 256.358,A -85,B 0,C 180,E1 -6413.511,E2 -6413.511} C_VEL
LIN {X 0,Y 490.811,Z 269.973,A -85,B 0,C 180,E1 -6413.889,E2 -6413.889} C_VEL
LIN {X 0,Y 490.592,Z 282.771,A -85,B 0,C 180,E1 -6414.424,E2 -6414.424} C_VEL
LIN {X 0,Y 490.23,Z 295.16,A -85,B 0,C 180,E1 -6415.133,E2 -6415.133} C_VEL
LIN {X 0,Y 489.783,Z 306.359,A -85,B 0,C 180,E1 -6415.955,E2 -6415.955} C_VEL
LIN {X 0,Y 489.445,Z 315.925,A -85,B 0,C 180,E1 -6416.828,E2 -6416.828} C_VEL
LIN {X 0,Y 489.08,Z 325.02,A -85,B 0,C 180,E1 -6417.842,E2 -6417.842} C_VEL
LIN {X 0,Y 488.8,Z 333.186,A -85,B 0,C 180,E1 -6418.958,E2 -6418.958} C_VEL
LIN {X 0,Y 488.49,Z 341.22,A -85,B 0,C 180,E1 -6420.32,E2 -6420.32} C_VEL
LIN {X 0,Y 488.29,Z 346.914,A -85,B 0,C 180,E1 -6421.534,E2 -6421.534} C_VEL
LIN {X 0,Y 488.132,Z 351.192,A -85,B 0,C 180,E1 -6422.678,E2 -6422.678} C_VEL
LIN {X 0,Y 487.994,Z 355.409,A -85,B 0,C 180,E1 -6424.172,E2 -6424.172} C_VEL
LIN {X 0,Y 487.905,Z 357.419,A -85,B 0,C 180,E1 -6425.183,E2 -6425.183} C_VEL
LIN {X 0,Y 487.826,Z 358.854,A -85,B 0,C 180,E1 -6426.219,E2 -6426.219} C_VEL
LIN {X 0,Y 487.833,Z 359.772,A -85,B 0,C 180,E1 -6427.594,E2 -6427.594} C_VEL
LIN {X 0,Y 487.826,Z 359.621,A -85,B 0,C 180,E1 -6428.926,E2 -6428.926} C_VEL
LIN {X 0,Y 487.885,Z 358.234,A -85,B 0,C 180,E1 -6430.409,E2 -6430.409} C_VEL
LIN {X 0,Y 488.034,Z 355.212,A -85,B 0,C 180,E1 -6432.039,E2 -6432.039} C_VEL
LIN {X 0,Y 488.142,Z 352.023,A -85,B 0,C 180,E1 -6433.196,E2 -6433.196} C_VEL
LIN {X 0,Y 488.299,Z 346.843,A -85,B 0,C 180,E1 -6434.608,E2 -6434.608} C_VEL
LIN {X 0,Y 488.541,Z 340.197,A -85,B 0,C 180,E1 -6435.996,E2 -6435.996} C_VEL
LIN {X 0,Y 488.831,Z 332.112,A -85,B 0,C 180,E1 -6437.33,E2 -6437.33} C_VEL
LIN {X 0,Y 489.201,Z 323.228,A -85,B 0,C 180,E1 -6438.493,E2 -6438.493} C_VEL
LIN {X 0,Y 489.627,Z 312.665,A -85,B 0,C 180,E1 -6439.61,E2 -6439.61} C_VEL
LIN {X 0,Y 489.995,Z 301.365,A -85,B 0,C 180,E1 -6440.554,E2 -6440.554} C_VEL
LIN {X 0,Y 490.457,Z 289.844,A -85,B 0,C 180,E1 -6441.31,E2 -6441.31} C_VEL
LIN {X 0,Y 490.79,Z 278.691,A -85,B 0,C 180,E1 -6441.877,E2 -6441.877} C_VEL
LIN {X 0,Y 490.962,Z 266.554,A -85,B 0,C 180,E1 -6442.334,E2 -6442.334} C_VEL
LIN {X 0,Y 491.161,Z 253.795,A -85,B 0,C 180,E1 -6442.643,E2 -6442.643} C_VEL
LIN {X 0,Y 491.746,Z 160.878,A -85,B 0,C 180,E1 -6444.051,E2 -6444.051} C_VEL
LIN {X 0,Y 489.438,Z 149.795,A -85,B 0,C 180,E1 -6444.315,E2 -6444.315} C_VEL
LIN {X 0,Y 489.564,Z 137.91,A -85,B 0,C 180,E1 -6446.652,E2 -6446.652} C_VEL
LIN {X 0,Y 488.753,Z 132.608,A -85,B 0,C 180,E1 -6447.766,E2 -6447.766} C_VEL
LIN {X 0,Y 488.725,Z 132.607,A -85,B 0,C 180,E1 -6450.73,E2 -6450.73} C_VEL
LIN {X 0,Y 488.738,Z 132.61,A -85,B 0,C 180,E1 -6453.528,E2 -6453.528} C_VEL
LIN {X 0,Y 488.674,Z 132.613,A -85,B 0,C 180,E1 -6456.254,E2 -6456.254} C_VEL
LIN {X 0,Y 488.75,Z 132.608,A -85,B 0,C 180,E1 -6459.176,E2 -6459.176} C_VEL
LIN {X 0,Y 488.751,Z 132.602,A -85,B 0,C 180,E1 -6461.633,E2 -6461.633} C_VEL
LIN {X 0,Y 488.763,Z 132.606,A -85,B 0,C 180,E1 -6465,E2 -6465} C_VEL
LIN {X 0,Y 488.809,Z 132.6,A -85,B 0,C 180,E1 -6468.388,E2 -6468.388} C_VEL
LIN {X 0,Y 488.784,Z 132.598,A -85,B 0,C 180,E1 -6471.734,E2 -6471.734} C_VEL
LIN {X 0,Y 488.82,Z 132.598,A -85,B 0,C 180,E1 -6474.224,E2 -6474.224} C_VEL
LIN {X 0,Y 488.947,Z 132.577,A -85,B 0,C 180,E1 -6477.529,E2 -6477.529} C_VEL
LIN {X 0,Y 488.946,Z 132.578,A -85,B 0,C 180,E1 -6480,E2 -6480} C_VEL
LIN {X 0,Y 488.945,Z 132.576,A -85,B 0,C 180,E1 -6482.472,E2 -6482.472} C_VEL
LIN {X 0,Y 488.814,Z 132.597,A -85,B 0,C 180,E1 -6485.777,E2 -6485.777} C_VEL
LIN {X 0,Y 488.759,Z 132.603,A -85,B 0,C 180,E1 -6488.268,E2 -6488.268} C_VEL
LIN {X 0,Y 488.779,Z 132.597,A -85,B 0,C 180,E1 -6491.614,E2 -6491.614} C_VEL
LIN {X 0,Y 488.718,Z 132.602,A -85,B 0,C 180,E1 -6495.002,E2 -6495.002} C_VEL
LIN {X 0,Y 488.68,Z 132.607,A -85,B 0,C 180,E1 -6498.445,E2 -6498.445} C_VEL
LIN {X 0,Y 488.681,Z 132.611,A -85,B 0,C 180,E1 -6501.072,E2 -6501.072} C_VEL
LIN {X 0,Y 488.661,Z 132.613,A -85,B 0,C 180,E1 -6503.748,E2 -6503.748} C_VEL
LIN {X 0,Y 488.672,Z 132.61,A -85,B 0,C 180,E1 -6506.477,E2 -6506.477} C_VEL
LIN {X 0,Y 488.664,Z 132.618,A -85,B 0,C 180,E1 -6509.275,E2 -6509.275} C_VEL
LIN {X 0,Y 488.695,Z 132.606,A -85,B 0,C 180,E1 -6512.148,E2 -6512.148} C_VEL
LIN {X 0,Y 488.717,Z 132.609,A -85,B 0,C 180,E1 -6515.116,E2 -6515.116} C_VEL
LIN {X 0,Y 488.679,Z 132.609,A -85,B 0,C 180,E1 -6518.201,E2 -6518.201} C_VEL
LIN {X 0,Y 488.698,Z 132.61,A -85,B 0,C 180,E1 -6520.341,E2 -6520.341} C_VEL
LIN {X 0,Y 488.678,Z 132.61,A -85,B 0,C 180,E1 -6523.656,E2 -6523.656} C_VEL
LIN {X 0,Y 488.68,Z 132.617,A -85,B 0,C 180,E1 -6526.344,E2 -6526.344} C_VEL
LIN {X 0,Y 488.708,Z 132.608,A -85,B 0,C 180,E1 -6529.673,E2 -6529.673} C_VEL
LIN {X 0,Y 488.675,Z 132.613,A -85,B 0,C 180,E1 -6532.84,E2 -6532.84} C_VEL
LIN {X 0,Y 488.735,Z 132.608,A -85,B 0,C 180,E1 -6535.887,E2 -6535.887} C_VEL
LIN {X 0,Y 488.696,Z 132.611,A -85,B 0,C 180,E1 -6538.82,E2 -6538.82} C_VEL
LIN {X 0,Y 488.718,Z 132.61,A -85,B 0,C 180,E1 -6541.669,E2 -6541.669} C_VEL
LIN {X 0,Y 488.782,Z 132.622,A -85,B 0,C 180,E1 -6544.274,E2 -6544.274} C_VEL
LIN {X 0,Y 490.507,Z 141.945,A -85,B 0,C 180,E1 -6545.898,E2 -6545.898} C_VEL
LIN {X 0,Y 490.435,Z 150.134,A -85,B 0,C 180,E1 -6547.237,E2 -6547.237} C_VEL
LIN {X 0,Y 489.838,Z 166.479,A -85,B 0,C 180,E1 -6549.858,E2 -6549.858} C_VEL
LIN {X 0,Y 489.461,Z 181.43,A -85,B 0,C 180,E1 -6552.234,E2 -6552.234} C_VEL
LIN {X 0,Y 489.189,Z 190.789,A -85,B 0,C 180,E1 -6553.71,E2 -6553.71} C_VEL
LIN {X 0,Y 491.672,Z 208.223,A -85,B 0,C 180,E1 -6554.065,E2 -6554.065} C_VEL
LIN {X 0,Y 491.027,Z 300.334,A -85,B 0,C 180,E1 -6555.467,E2 -6555.467} C_VEL
LIN {X 0,Y 490.679,Z 313.328,A -85,B 0,C 180,E1 -6555.827,E2 -6555.827} C_VEL
LIN {X 0,Y 490.324,Z 325.382,A -85,B 0,C 180,E1 -6556.319,E2 -6556.319} C_VEL
LIN {X 0,Y 489.92,Z 337.112,A -85,B 0,C 180,E1 -6556.963,E2 -6556.963} C_VEL
LIN {X 0,Y 489.479,Z 348.541,A -85,B 0,C 180,E1 -6557.773,E2 -6557.773} C_VEL
LIN {X 0,Y 489.081,Z 359.116,A -85,B 0,C 180,E1 -6558.709,E2 -6558.709} C_VEL
LIN {X 0,Y 488.743,Z 367.766,A -85,B 0,C 180,E1 -6559.644,E2 -6559.644} C_VEL
LIN {X 0,Y 488.466,Z 375.748,A -85,B 0,C 180,E1 -6560.684,E2 -6560.684} C_VEL
LIN {X 0,Y 488.234,Z 383.552,A -85,B 0,C 180,E1 -6561.931,E2 -6561.931} C_VEL
LIN {X 0,Y 488.092,Z 388.893,A -85,B 0,C 180,E1 -6562.969,E2 -6562.969} C_VEL
LIN {X 0,Y 487.997,Z 394.077,A -85,B 0,C 180,E1 -6564.214,E2 -6564.214} C_VEL
LIN {X 0,Y 487.919,Z 398.101,A -85,B 0,C 180,E1 -6565.456,E2 -6565.456} C_VEL
LIN {X 0,Y 487.978,Z 401.081,A -85,B 0,C 180,E1 -6566.697,E2 -6566.697} C_VEL
LIN {X 0,Y 487.937,Z 402.499,A -85,B 0,C 180,E1 -6567.523,E2 -6567.523} C_VEL
LIN {X 0,Y 487.893,Z 403.512,A -85,B 0,C 180,E1 -6568.349,E2 -6568.349} C_VEL
LIN {X 0,Y 487.834,Z 404.359,A -85,B 0,C 180,E1 -6570,E2 -6570} C_VEL
LIN {X 0,Y 487.893,Z 403.543,A -85,B 0,C 180,E1 -6571.65,E2 -6571.65} C_VEL
LIN {X 0,Y 487.937,Z 402.547,A -85,B 0,C 180,E1 -6572.476,E2 -6572.476} C_VEL
LIN {X 0,Y 487.978,Z 401.142,A -85,B 0,C 180,E1 -6573.302,E2 -6573.302} C_VEL
LIN {X 0,Y 487.919,Z 398.182,A -85,B 0,C 180,E1 -6574.543,E2 -6574.543} C_VEL
LIN {X 0,Y 488.003,Z 394.178,A -85,B 0,C 180,E1 -6575.785,E2 -6575.785} C_VEL
LIN {X 0,Y 488.172,Z 388.011,A -85,B 0,C 180,E1 -6577.236,E2 -6577.236} C_VEL
LIN {X 0,Y 488.317,Z 381.273,A -85,B 0,C 180,E1 -6578.483,E2 -6578.483} C_VEL
LIN {X 0,Y 488.569,Z 372.915,A -85,B 0,C 180,E1 -6579.73,E2 -6579.73} C_VEL
LIN {X 0,Y 488.929,Z 364.328,A -85,B 0,C 180,E1 -6580.769,E2 -6580.769} C_VEL
LIN {X 0,Y 489.313,Z 353.737,A -85,B 0,C 180,E1 -6581.809,E2 -6581.809} C_VEL
LIN {X 0,Y 489.711,Z 342.435,A -85,B 0,C 180,E1 -6582.699,E2 -6582.699} C_VEL
LIN {X 0,Y 490.102,Z 331.667,A -85,B 0,C 180,E1 -6583.369,E2 -6583.369} C_VEL
LIN {X 0,Y 490.47,Z 319.69,A -85,B 0,C 180,E1 -6583.94,E2 -6583.94} C_VEL
LIN {X 0,Y 490.836,Z 306.772,A -85,B 0,C 180,E1 -6584.379,E2 -6584.379} C_VEL
LIN {X 0,Y 491.084,Z 293.137,A -85,B 0,C 180,E1 -6584.662,E2 -6584.662} C_VEL
LIN {X 0,Y 491.549,Z 207.324,A -85,B 0,C 180,E1 -6585.945,E2 -6585.945} C_VEL
LIN {X 0,Y 489.236,Z 191.366,A -85,B 0,C 180,E1 -6586.267,E2 -6586.267} C_VEL
LIN {X 0,Y 489.854,Z 171.219,A -85,B 0,C 180,E1 -6589.485,E2 -6589.485} C_VEL
LIN {X 0,Y 490.568,Z 151.039,A -85,B 0,C 180,E1 -6592.756,E2 -6592.756} C_VEL
LIN {X 0,Y 490.768,Z 142.94,A -85,B 0,C 180,E1 -6594.087,E2 -6594.087} C_VEL
LIN {X 0,Y 488.778,Z 132.604,A -85,B 0,C 180,E1 -6595.954,E2 -6595.954} C_VEL
LIN {X 0,Y 488.73,Z 132.607,A -85,B 0,C 180,E1 -6598.694,E2 -6598.694} C_VEL
LIN {X 0,Y 488.693,Z 132.607,A -85,B 0,C 180,E1 -6601.179,E2 -6601.179} C_VEL
LIN {X 0,Y 488.731,Z 132.608,A -85,B 0,C 180,E1 -6604.112,E2 -6604.112} C_VEL
LIN {X 0,Y 488.68,Z 132.609,A -85,B 0,C 180,E1 -6607.158,E2 -6607.158} C_VEL
LIN {X 0,Y 488.719,Z 132.606,A -85,B 0,C 180,E1 -6610.344,E2 -6610.344} C_VEL
LIN {X 0,Y 488.684,Z 132.614,A -85,B 0,C 180,E1 -6613.654,E2 -6613.654} C_VEL
LIN {X 0,Y 488.685,Z 132.609,A -85,B 0,C 180,E1 -6616.345,E2 -6616.345} C_VEL
LIN {X 0,Y 488.733,Z 132.61,A -85,B 0,C 180,E1 -6619.676,E2 -6619.676} C_VEL
LIN {X 0,Y 488.679,Z 132.609,A -85,B 0,C 180,E1 -6622.841,E2 -6622.841} C_VEL
LIN {X 0,Y 488.723,Z 132.607,A -85,B 0,C 180,E1 -6625.886,E2 -6625.886} C_VEL
LIN {X 0,Y 488.69,Z 132.608,A -85,B 0,C 180,E1 -6628.82,E2 -6628.82} C_VEL
LIN {X 0,Y 488.743,Z 132.605,A -85,B 0,C 180,E1 -6631.671,E2 -6631.671} C_VEL
LIN {X 0,Y 488.746,Z 132.6,A -85,B 0,C 180,E1 -6634.444,E2 -6634.444} C_VEL
LIN {X 0,Y 488.722,Z 132.609,A -85,B 0,C 180,E1 -6637.153,E2 -6637.153} C_VEL
LIN {X 0,Y 488.723,Z 132.604,A -85,B 0,C 180,E1 -6639.81,E2 -6639.81} C_VEL
LIN {X 0,Y 488.714,Z 132.604,A -85,B 0,C 180,E1 -6642.422,E2 -6642.422} C_VEL
LIN {X 0,Y 488.761,Z 132.604,A -85,B 0,C 180,E1 -6644.999,E2 -6644.999} C_VEL
LIN {X 0,Y 488.804,Z 132.593,A -85,B 0,C 180,E1 -6648.387,E2 -6648.387} C_VEL
LIN {X 0,Y 488.816,Z 132.592,A -85,B 0,C 180,E1 -6651.733,E2 -6651.733} C_VEL
LIN {X 0,Y 488.847,Z 132.588,A -85,B 0,C 180,E1 -6654.224,E2 -6654.224} C_VEL
LIN {X 0,Y 488.96,Z 132.574,A -85,B 0,C 180,E1 -6657.528,E2 -6657.528} C_VEL
LIN {X 0,Y 488.953,Z 132.583,A -85,B 0,C 180,E1 -6660.823,E2 -6660.823} C_VEL
LIN {X 0,Y 488.96,Z 132.577,A -85,B 0,C 180,E1 -6662.471,E2 -6662.471} C_VEL
LIN {X 0,Y 488.847,Z 132.587,A -85,B 0,C 180,E1 -6665.775,E2 -6665.775} C_VEL
LIN {X 0,Y 488.816,Z 132.594,A -85,B 0,C 180,E1 -6668.266,E2 -6668.266} C_VEL
LIN {X 0,Y 488.803,Z 132.593,A -85,B 0,C 180,E1 -6671.612,E2 -6671.612} C_VEL
LIN {X 0,Y 488.762,Z 132.6,A -85,B 0,C 180,E1 -6675,E2 -6675} C_VEL
LIN {X 0,Y 488.752,Z 132.608,A -85,B 0,C 180,E1 -6678.442,E2 -6678.442} C_VEL
LIN {X 0,Y 488.703,Z 132.606,A -85,B 0,C 180,E1 -6681.07,E2 -6681.07} C_VEL
LIN {X 0,Y 488.686,Z 132.609,A -85,B 0,C 180,E1 -6683.745,E2 -6683.745} C_VEL
LIN {X 0,Y 488.795,Z 132.595,A -85,B 0,C 180,E1 -6686.945,E2 -6686.945} C_VEL
LIN {X 0,Y 488.706,Z 132.611,A -85,B 0,C 180,E1 -6690.363,E2 -6690.363} C_VEL
LIN {X 0,Y 488.731,Z 132.603,A -85,B 0,C 180,E1 -6693.484,E2 -6693.484} C_VEL
LIN {X 0,Y 488.684,Z 132.612,A -85,B 0,C 180,E1 -6696.355,E2 -6696.355} C_VEL
LIN {X 0,Y 488.744,Z 132.6,A -85,B 0,C 180,E1 -6699.249,E2 -6699.249} C_VEL
LIN {X 0,Y 488.727,Z 132.604,A -85,B 0,C 180,E1 -6702.521,E2 -6702.521} C_VEL
LIN {X 0,Y 488.707,Z 132.605,A -85,B 0,C 180,E1 -6705.199,E2 -6705.199} C_VEL
LIN {X 0,Y 488.727,Z 132.606,A -85,B 0,C 180,E1 -6707.479,E2 -6707.479} C_VEL
LIN {X 0,Y 488.744,Z 132.6,A -85,B 0,C 180,E1 -6710.75,E2 -6710.75} C_VEL
LIN {X 0,Y 488.68,Z 132.615,A -85,B 0,C 180,E1 -6713.869,E2 -6713.869} C_VEL
LIN {X 0,Y 488.734,Z 132.602,A -85,B 0,C 180,E1 -6716.877,E2 -6716.877} C_VEL
LIN {X 0,Y 488.719,Z 132.609,A -85,B 0,C 180,E1 -6719.781,E2 -6719.781} C_VEL
LIN {X 0,Y 488.794,Z 132.596,A -85,B 0,C 180,E1 -6723.055,E2 -6723.055} C_VEL
LIN {X 0,Y 488.742,Z 132.601,A -85,B 0,C 180,E1 -6724.346,E2 -6724.346} C_VEL
LIN {X 0,Y 488.094,Z 132.685,A -85,B 0,C 180,E1 -6725.034,E2 -6725.034} C_VEL
LIN {X 0,Y 485.224,Z 133.043,A -85,B 0,C 180,E1 -6726.15,E2 -6726.15} C_VEL
LIN {X 0,Y 482.778,Z 133.349,A -85,B 0,C 180,E1 -6727.05,E2 -6727.05} C_VEL
LIN {X 0,Y 481.721,Z 133.48,A -85,B 0,C 180,E1 -6727.745,E2 -6727.745} C_VEL
LIN {X 0,Y 481.633,Z 133.488,A -85,B 0,C 180,E1 -6727.981,E2 -6727.981} C_VEL
LIN {X 0,Y 481.703,Z 133.477,A -85,B 0,C 180,E1 -6730.393,E2 -6730.393} C_VEL
LIN {X 0,Y 481.687,Z 133.483,A -85,B 0,C 180,E1 -6733.034,E2 -6733.034} C_VEL
LIN {X 0,Y 481.69,Z 133.483,A -85,B 0,C 180,E1 -6735.639,E2 -6735.639} C_VEL
LIN {X 0,Y 481.747,Z 133.472,A -85,B 0,C 180,E1 -6738.215,E2 -6738.215} C_VEL
LIN {X 0,Y 481.759,Z 133.473,A -85,B 0,C 180,E1 -6741.612,E2 -6741.612} C_VEL
LIN {X 0,Y 481.816,Z 133.463,A -85,B 0,C 180,E1 -6744.14,E2 -6744.14} C_VEL
LIN {X 0,Y 481.926,Z 133.452,A -85,B 0,C 180,E1 -6747.493,E2 -6747.493} C_VEL
LIN {X 0,Y 481.902,Z 133.459,A -85,B 0,C 180,E1 -6750.836,E2 -6750.836} C_VEL
LIN {X 0,Y 481.926,Z 133.452,A -85,B 0,C 180,E1 -6752.508,E2 -6752.508} C_VEL
LIN {X 0,Y 481.817,Z 133.463,A -85,B 0,C 180,E1 -6755.861,E2 -6755.861} C_VEL
LIN {X 0,Y 481.761,Z 133.473,A -85,B 0,C 180,E1 -6758.389,E2 -6758.389} C_VEL
LIN {X 0,Y 481.748,Z 133.472,A -85,B 0,C 180,E1 -6761.785,E2 -6761.785} C_VEL
LIN {X 0,Y 481.742,Z 133.478,A -85,B 0,C 180,E1 -6765.225,E2 -6765.225} C_VEL
LIN {X 0,Y 481.764,Z 133.538,A -85,B 0,C 180,E1 -6768.201,E2 -6768.201} C_VEL
LIN {X 0,Y 482.605,Z 139.961,A -85,B 0,C 180,E1 -6769.569,E2 -6769.569} C_VEL
LIN {X 0,Y 482.423,Z 149.706,A -85,B 0,C 180,E1 -6771.567,E2 -6771.567} C_VEL
LIN {X 0,Y 485.023,Z 163.721,A -85,B 0,C 180,E1 -6771.882,E2 -6771.882} C_VEL
LIN {X 0,Y 484.209,Z 256.846,A -85,B 0,C 180,E1 -6773.312,E2 -6773.312} C_VEL
LIN {X 0,Y 483.939,Z 270.296,A -85,B 0,C 180,E1 -6773.692,E2 -6773.692} C_VEL
LIN {X 0,Y 483.695,Z 283.105,A -85,B 0,C 180,E1 -6774.235,E2 -6774.235} C_VEL
LIN {X 0,Y 483.331,Z 295.302,A -85,B 0,C 180,E1 -6774.941,E2 -6774.941} C_VEL
LIN {X 0,Y 482.849,Z 306.545,A -85,B 0,C 180,E1 -6775.775,E2 -6775.775} C_VEL
LIN {X 0,Y 482.46,Z 316.807,A -85,B 0,C 180,E1 -6776.729,E2 -6776.729} C_VEL
LIN {X 0,Y 482.049,Z 326.194,A -85,B 0,C 180,E1 -6777.811,E2 -6777.811} C_VEL
LIN {X 0,Y 481.714,Z 335.039,A -85,B 0,C 180,E1 -6779.071,E2 -6779.071} C_VEL
LIN {X 0,Y 481.448,Z 341.18,A -85,B 0,C 180,E1 -6780.145,E2 -6780.145} C_VEL
LIN {X 0,Y 481.232,Z 347.359,A -85,B 0,C 180,E1 -6781.474,E2 -6781.474} C_VEL
LIN {X 0,Y 481.059,Z 351.904,A -85,B 0,C 180,E1 -6782.722,E2 -6782.722} C_VEL
LIN {X 0,Y 480.9,Z 355.984,A -85,B 0,C 180,E1 -6784.24,E2 -6784.24} C_VEL
LIN {X 0,Y 480.779,Z 358.684,A -85,B 0,C 180,E1 -6785.784,E2 -6785.784} C_VEL
LIN {X 0,Y 480.752,Z 359.732,A -85,B 0,C 180,E1 -6786.825,E2 -6786.825} C_VEL
LIN {X 0,Y 480.748,Z 360.154,A -85,B 0,C 180,E1 -6787.879,E2 -6787.879} C_VEL
LIN {X 0,Y 480.737,Z 359.795,A -85,B 0,C 180,E1 -6789.212,E2 -6789.212} C_VEL
LIN {X 0,Y 480.815,Z 358.448,A -85,B 0,C 180,E1 -6790.53,E2 -6790.53} C_VEL
LIN {X 0,Y 480.962,Z 355.198,A -85,B 0,C 180,E1 -6792.235,E2 -6792.235} C_VEL
LIN {X 0,Y 481.096,Z 350.503,A -85,B 0,C 180,E1 -6793.832,E2 -6793.832} C_VEL
LIN {X 0,Y 481.312,Z 344.776,A -85,B 0,C 180,E1 -6795.258,E2 -6795.258} C_VEL
LIN {X 0,Y 481.619,Z 337.255,A -85,B 0,C 180,E1 -6796.699,E2 -6796.699} C_VEL
LIN {X 0,Y 481.962,Z 329.585,A -85,B 0,C 180,E1 -6797.874,E2 -6797.874} C_VEL
LIN {X 0,Y 482.358,Z 320.243,A -85,B 0,C 180,E1 -6799.031,E2 -6799.031} C_VEL
LIN {X 0,Y 482.797,Z 310.195,A -85,B 0,C 180,E1 -6800.036,E2 -6800.036} C_VEL
LIN {X 0,Y 483.194,Z 299.687,A -85,B 0,C 180,E1 -6800.885,E2 -6800.885} C_VEL
LIN {X 0,Y 483.624,Z 288.24,A -85,B 0,C 180,E1 -6801.617,E2 -6801.617} C_VEL
LIN {X 0,Y 483.975,Z 275.377,A -85,B 0,C 180,E1 -6802.233,E2 -6802.233} C_VEL
LIN {X 0,Y 484.146,Z 263.039,A -85,B 0,C 180,E1 -6802.655,E2 -6802.655} C_VEL
LIN {X 0,Y 484.344,Z 250.039,A -85,B 0,C 180,E1 -6802.926,E2 -6802.926} C_VEL
LIN {X 0,Y 484.996,Z 161.969,A -85,B 0,C 180,E1 -6804.272,E2 -6804.272} C_VEL
LIN {X 0,Y 482.479,Z 150.132,A -85,B 0,C 180,E1 -6804.555,E2 -6804.555} C_VEL
LIN {X 0,Y 482.618,Z 139.576,A -85,B 0,C 180,E1 -6806.653,E2 -6806.653} C_VEL
LIN {X 0,Y 481.694,Z 133.487,A -85,B 0,C 180,E1 -6807.924,E2 -6807.924} C_VEL
LIN {X 0,Y 481.702,Z 133.485,A -85,B 0,C 180,E1 -6811.219,E2 -6811.219} C_VEL
LIN {X 0,Y 481.677,Z 133.486,A -85,B 0,C 180,E1 -6814.042,E2 -6814.042} C_VEL
LIN {X 0,Y 481.677,Z 133.489,A -85,B 0,C 180,E1 -6816.813,E2 -6816.813} C_VEL
LIN {X 0,Y 481.698,Z 133.482,A -85,B 0,C 180,E1 -6819.503,E2 -6819.503} C_VEL
LIN {X 0,Y 481.692,Z 133.481,A -85,B 0,C 180,E1 -6822.158,E2 -6822.158} C_VEL
LIN {X 0,Y 481.745,Z 133.48,A -85,B 0,C 180,E1 -6824.776,E2 -6824.776} C_VEL
LIN {X 0,Y 481.755,Z 133.477,A -85,B 0,C 180,E1 -6828.216,E2 -6828.216} C_VEL
LIN {X 0,Y 481.74,Z 133.476,A -85,B 0,C 180,E1 -6831.612,E2 -6831.612} C_VEL
LIN {X 0,Y 481.781,Z 133.474,A -85,B 0,C 180,E1 -6834.14,E2 -6834.14} C_VEL
LIN {X 0,Y 481.913,Z 133.453,A -85,B 0,C 180,E1 -6837.493,E2 -6837.493} C_VEL
LIN {X 0,Y 481.915,Z 133.453,A -85,B 0,C 180,E1 -6840,E2 -6840} C_VEL
LIN {X 0,Y 481.911,Z 133.452,A -85,B 0,C 180,E1 -6842.508,E2 -6842.508} C_VEL
LIN {X 0,Y 481.776,Z 133.475,A -85,B 0,C 180,E1 -6845.861,E2 -6845.861} C_VEL
LIN {X 0,Y 481.717,Z 133.479,A -85,B 0,C 180,E1 -6848.39,E2 -6848.39} C_VEL
LIN {X 0,Y 481.73,Z 133.477,A -85,B 0,C 180,E1 -6851.786,E2 -6851.786} C_VEL
LIN {X 0,Y 481.694,Z 133.478,A -85,B 0,C 180,E1 -6855.226,E2 -6855.226} C_VEL
LIN {X 0,Y 481.626,Z 133.486,A -85,B 0,C 180,E1 -6858.726,E2 -6858.726} C_VEL
LIN {X 0,Y 481.625,Z 133.494,A -85,B 0,C 180,E1 -6861.396,E2 -6861.396} C_VEL
LIN {X 0,Y 481.622,Z 133.487,A -85,B 0,C 180,E1 -6864.116,E2 -6864.116} C_VEL
LIN {X 0,Y 481.646,Z 133.49,A -85,B 0,C 180,E1 -6867.114,E2 -6867.114} C_VEL
LIN {X 0,Y 481.604,Z 133.492,A -85,B 0,C 180,E1 -6869.747,E2 -6869.747} C_VEL
LIN {X 0,Y 481.654,Z 133.486,A -85,B 0,C 180,E1 -6872.676,E2 -6872.676} C_VEL
LIN {X 0,Y 481.635,Z 133.487,A -85,B 0,C 180,E1 -6875.71,E2 -6875.71} C_VEL
LIN {X 0,Y 481.67,Z 133.487,A -85,B 0,C 180,E1 -6878.86,E2 -6878.86} C_VEL
LIN {X 0,Y 481.62,Z 133.49,A -85,B 0,C 180,E1 -6882.164,E2 -6882.164} C_VEL
LIN {X 0,Y 481.658,Z 133.489,A -85,B 0,C 180,E1 -6884.458,E2 -6884.458} C_VEL
LIN {X 0,Y 481.634,Z 133.49,A -85,B 0,C 180,E1 -6887.837,E2 -6887.837} C_VEL
LIN {X 0,Y 481.671,Z 133.484,A -85,B 0,C 180,E1 -6891.14,E2 -6891.14} C_VEL
LIN {X 0,Y 481.666,Z 133.486,A -85,B 0,C 180,E1 -6894.796,E2 -6894.796} C_VEL
LIN {X 0,Y 481.677,Z 133.486,A -85,B 0,C 180,E1 -6897.326,E2 -6897.326} C_VEL
LIN {X 0,Y 481.677,Z 133.489,A -85,B 0,C 180,E1 -6900.258,E2 -6900.258} C_VEL
LIN {X 0,Y 481.691,Z 133.484,A -85,B 0,C 180,E1 -6903.108,E2 -6903.108} C_VEL
LIN {X 0,Y 481.734,Z 133.61,A -85,B 0,C 180,E1 -6904.09,E2 -6904.09} C_VEL
LIN {X 0,Y 483.521,Z 143,A -85,B 0,C 180,E1 -6905.756,E2 -6905.756} C_VEL
LIN {X 0,Y 483.629,Z 147.893,A -85,B 0,C 180,E1 -6906.576,E2 -6906.576} C_VEL
LIN {X 0,Y 482.908,Z 166.159,A -85,B 0,C 180,E1 -6909.556,E2 -6909.556} C_VEL
LIN {X 0,Y 482.43,Z 182.465,A -85,B 0,C 180,E1 -6912.186,E2 -6912.186} C_VEL
LIN {X 0,Y 482.214,Z 190.455,A -85,B 0,C 180,E1 -6913.466,E2 -6913.466} C_VEL
LIN {X 0,Y 484.834,Z 209.099,A -85,B 0,C 180,E1 -6913.849,E2 -6913.849} C_VEL
LIN {X 0,Y 484.16,Z 300.032,A -85,B 0,C 180,E1 -6915.257,E2 -6915.257} C_VEL
LIN {X 0,Y 483.801,Z 313.002,A -85,B 0,C 180,E1 -6915.622,E2 -6915.622} C_VEL
LIN {X 0,Y 483.398,Z 325.042,A -85,B 0,C 180,E1 -6916.119,E2 -6916.119} C_VEL
LIN {X 0,Y 482.964,Z 336.443,A -85,B 0,C 180,E1 -6916.75,E2 -6916.75} C_VEL
LIN {X 0,Y 482.565,Z 347.286,A -85,B 0,C 180,E1 -6917.52,E2 -6917.52} C_VEL
LIN {X 0,Y 482.135,Z 357.688,A -85,B 0,C 180,E1 -6918.437,E2 -6918.437} C_VEL
LIN {X 0,Y 481.706,Z 367.42,A -85,B 0,C 180,E1 -6919.492,E2 -6919.492} C_VEL
LIN {X 0,Y 481.429,Z 375.408,A -85,B 0,C 180,E1 -6920.547,E2 -6920.547} C_VEL
LIN {X 0,Y 481.155,Z 383.215,A -85,B 0,C 180,E1 -6921.812,E2 -6921.812} C_VEL
LIN {X 0,Y 480.966,Z 390.404,A -85,B 0,C 180,E1 -6923.286,E2 -6923.286} C_VEL
LIN {X 0,Y 480.919,Z 395.196,A -85,B 0,C 180,E1 -6924.549,E2 -6924.549} C_VEL
LIN {X 0,Y 480.83,Z 398.858,A -85,B 0,C 180,E1 -6925.808,E2 -6925.808} C_VEL
LIN {X 0,Y 480.901,Z 400.754,A -85,B 0,C 180,E1 -6926.648,E2 -6926.648} C_VEL
LIN {X 0,Y 480.85,Z 402.173,A -85,B 0,C 180,E1 -6927.486,E2 -6927.486} C_VEL
LIN {X 0,Y 480.824,Z 403.189,A -85,B 0,C 180,E1 -6928.324,E2 -6928.324} C_VEL
LIN {X 0,Y 480.757,Z 404.036,A -85,B 0,C 180,E1 -6930,E2 -6930} C_VEL
LIN {X 0,Y 480.824,Z 403.22,A -85,B 0,C 180,E1 -6931.675,E2 -6931.675} C_VEL
LIN {X 0,Y 480.85,Z 402.222,A -85,B 0,C 180,E1 -6932.513,E2 -6932.513} C_VEL
LIN {X 0,Y 480.9,Z 400.816,A -85,B 0,C 180,E1 -6933.351,E2 -6933.351} C_VEL
LIN {X 0,Y 480.837,Z 397.853,A -85,B 0,C 180,E1 -6934.61,E2 -6934.61} C_VEL
LIN {X 0,Y 480.905,Z 393.843,A -85,B 0,C 180,E1 -6935.871,E2 -6935.871} C_VEL
LIN {X 0,Y 481.095,Z 387.668,A -85,B 0,C 180,E1 -6937.343,E2 -6937.343} C_VEL
LIN {X 0,Y 481.267,Z 380.921,A -85,B 0,C 180,E1 -6938.608,E2 -6938.608} C_VEL
LIN {X 0,Y 481.524,Z 372.551,A -85,B 0,C 180,E1 -6939.874,E2 -6939.874} C_VEL
LIN {X 0,Y 481.915,Z 363.946,A -85,B 0,C 180,E1 -6940.928,E2 -6940.928} C_VEL
LIN {X 0,Y 482.316,Z 353.554,A -85,B 0,C 180,E1 -6941.963,E2 -6941.963} C_VEL
LIN {X 0,Y 482.712,Z 343.097,A -85,B 0,C 180,E1 -6942.806,E2 -6942.806} C_VEL
LIN {X 0,Y 483.174,Z 331.219,A -85,B 0,C 180,E1 -6943.564,E2 -6943.564} C_VEL
LIN {X 0,Y 483.572,Z 319.197,A -85,B 0,C 180,E1 -6944.143,E2 -6944.143} C_VEL
LIN {X 0,Y 483.971,Z 306.214,A -85,B 0,C 180,E1 -6944.587,E2 -6944.587} C_VEL
LIN {X 0,Y 484.212,Z 292.357,A -85,B 0,C 180,E1 -6944.875,E2 -6944.875} C_VEL
LIN {X 0,Y 484.651,Z 207.794,A -85,B 0,C 180,E1 -6946.162,E2 -6946.162} C_VEL
LIN {X 0,Y 482.212,Z 191.026,A -85,B 0,C 180,E1 -6946.511,E2 -6946.511} C_VEL
LIN {X 0,Y 482.86,Z 172.245,A -85,B 0,C 180,E1 -6949.558,E2 -6949.558} C_VEL
LIN {X 0,Y 483.697,Z 150.703,A -85,B 0,C 180,E1 -6953.097,E2 -6953.097} C_VEL
LIN {X 0,Y 483.783,Z 143.954,A -85,B 0,C 180,E1 -6954.229,E2 -6954.229} C_VEL
LIN {X 0,Y 481.727,Z 133.482,A -85,B 0,C 180,E1 -6956.13,E2 -6956.13} C_VEL
LIN {X 0,Y 481.677,Z 133.484,A -85,B 0,C 180,E1 -6958.902,E2 -6958.902} C_VEL
LIN {X 0,Y 481.658,Z 133.491,A -85,B 0,C 180,E1 -6962.189,E2 -6962.189} C_VEL
LIN {X 0,Y 481.689,Z 133.48,A -85,B 0,C 180,E1 -6964.682,E2 -6964.682} C_VEL
LIN {X 0,Y 481.655,Z 133.49,A -85,B 0,C 180,E1 -6968.007,E2 -6968.007} C_VEL
LIN {X 0,Y 481.656,Z 133.483,A -85,B 0,C 180,E1 -6971.041,E2 -6971.041} C_VEL
LIN {X 0,Y 481.654,Z 133.484,A -85,B 0,C 180,E1 -6974.457,E2 -6974.457} C_VEL
LIN {X 0,Y 481.648,Z 133.491,A -85,B 0,C 180,E1 -6977.839,E2 -6977.839} C_VEL
LIN {X 0,Y 481.661,Z 133.482,A -85,B 0,C 180,E1 -6980.653,E2 -6980.653} C_VEL
LIN {X 0,Y 481.627,Z 133.492,A -85,B 0,C 180,E1 -6983.376,E2 -6983.376} C_VEL
LIN {X 0,Y 481.676,Z 133.481,A -85,B 0,C 180,E1 -6986.327,E2 -6986.327} C_VEL
LIN {X 0,Y 481.649,Z 133.492,A -85,B 0,C 180,E1 -6989.417,E2 -6989.417} C_VEL
LIN {X 0,Y 481.699,Z 133.478,A -85,B 0,C 180,E1 -6992.168,E2 -6992.168} C_VEL
LIN {X 0,Y 481.716,Z 133.479,A -85,B 0,C 180,E1 -6994.969,E2 -6994.969} C_VEL
LIN {X 0,Y 481.648,Z 133.487,A -85,B 0,C 180,E1 -6997.704,E2 -6997.704} C_VEL
LIN {X 0,Y 481.703,Z 133.477,A -85,B 0,C 180,E1 -7000.393,E2 -7000.393} C_VEL
LIN {X 0,Y 481.678,Z 133.487,A -85,B 0,C 180,E1 -7003.033,E2 -7003.033} C_VEL
LIN {X 0,Y 481.688,Z 133.481,A -85,B 0,C 180,E1 -7005.638,E2 -7005.638} C_VEL
LIN {X 0,Y 481.75,Z 133.472,A -85,B 0,C 180,E1 -7008.215,E2 -7008.215} C_VEL
LIN {X 0,Y 481.761,Z 133.471,A -85,B 0,C 180,E1 -7011.611,E2 -7011.611} C_VEL
LIN {X 0,Y 481.807,Z 133.464,A -85,B 0,C 180,E1 -7014.139,E2 -7014.139} C_VEL
LIN {X 0,Y 481.927,Z 133.451,A -85,B 0,C 180,E1 -7017.492,E2 -7017.492} C_VEL
LIN {X 0,Y 481.904,Z 133.461,A -85,B 0,C 180,E1 -7020.835,E2 -7020.835} C_VEL
LIN {X 0,Y 481.927,Z 133.454,A -85,B 0,C 180,E1 -7022.507,E2 -7022.507} C_VEL
LIN {X 0,Y 481.807,Z 133.464,A -85,B 0,C 180,E1 -7025.86,E2 -7025.86} C_VEL
LIN {X 0,Y 481.761,Z 133.474,A -85,B 0,C 180,E1 -7028.388,E2 -7028.388} C_VEL
LIN {X 0,Y 481.748,Z 133.472,A -85,B 0,C 180,E1 -7031.784,E2 -7031.784} C_VEL
LIN {X 0,Y 481.741,Z 133.473,A -85,B 0,C 180,E1 -7035.224,E2 -7035.224} C_VEL
LIN {X 0,Y 481.709,Z 133.481,A -85,B 0,C 180,E1 -7038.721,E2 -7038.721} C_VEL
LIN {X 0,Y 481.642,Z 133.485,A -85,B 0,C 180,E1 -7041.394,E2 -7041.394} C_VEL
LIN {X 0,Y 481.671,Z 133.486,A -85,B 0,C 180,E1 -7044.113,E2 -7044.113} C_VEL
LIN {X 0,Y 481.748,Z 133.472,A -85,B 0,C 180,E1 -7047.14,E2 -7047.14} C_VEL
LIN {X 0,Y 481.675,Z 133.483,A -85,B 0,C 180,E1 -7049.741,E2 -7049.741} C_VEL
LIN {X 0,Y 481.669,Z 133.484,A -85,B 0,C 180,E1 -7052.674,E2 -7052.674} C_VEL
LIN {X 0,Y 481.638,Z 133.488,A -85,B 0,C 180,E1 -7055.709,E2 -7055.709} C_VEL
LIN {X 0,Y 481.715,Z 133.477,A -85,B 0,C 180,E1 -7059.354,E2 -7059.354} C_VEL
LIN {X 0,Y 481.669,Z 133.487,A -85,B 0,C 180,E1 -7062.158,E2 -7062.158} C_VEL
LIN {X 0,Y 481.655,Z 133.485,A -85,B 0,C 180,E1 -7064.457,E2 -7064.457} C_VEL
LIN {X 0,Y 481.683,Z 133.48,A -85,B 0,C 180,E1 -7066.846,E2 -7066.846} C_VEL
LIN {X 0,Y 481.688,Z 133.484,A -85,B 0,C 180,E1 -7070.061,E2 -7070.061} C_VEL
LIN {X 0,Y 481.624,Z 133.489,A -85,B 0,C 180,E1 -7073.253,E2 -7073.253} C_VEL
LIN {X 0,Y 481.704,Z 133.478,A -85,B 0,C 180,E1 -7076.33,E2 -7076.33} C_VEL
LIN {X 0,Y 481.647,Z 133.49,A -85,B 0,C 180,E1 -7079.417,E2 -7079.417} C_VEL
LIN {X 0,Y 481.697,Z 133.479,A -85,B 0,C 180,E1 -7082.168,E2 -7082.168} C_VEL
LIN {X 0,Y 481.713,Z 133.478,A -85,B 0,C 180,E1 -7084.97,E2 -7084.97} C_VEL
LIN {X 0,Y 481.633,Z 133.488,A -85,B 0,C 180,E1 -7087.981,E2 -7087.981} C_VEL
LIN {X 0,Y 480.965,Z 133.57,A -85,B 0,C 180,E1 -7088.679,E2 -7088.679} C_VEL
LIN {X 0,Y 478.138,Z 133.927,A -85,B 0,C 180,E1 -7089.813,E2 -7089.813} C_VEL
LIN {X 0,Y 475.753,Z 134.227,A -85,B 0,C 180,E1 -7090.727,E2 -7090.727} C_VEL
LIN {X 0,Y 474.733,Z 134.353,A -85,B 0,C 180,E1 -7091.433,E2 -7091.433} C_VEL
LIN {X 0,Y 474.651,Z 134.36,A -85,B 0,C 180,E1 -7091.672,E2 -7091.672} C_VEL
LIN {X 0,Y 474.696,Z 134.351,A -85,B 0,C 180,E1 -7094.545,E2 -7094.545} C_VEL
LIN {X 0,Y 474.7,Z 134.35,A -85,B 0,C 180,E1 -7098.038,E2 -7098.038} C_VEL
LIN {X 0,Y 474.725,Z 134.351,A -85,B 0,C 180,E1 -7101.487,E2 -7101.487} C_VEL
LIN {X 0,Y 474.778,Z 134.34,A -85,B 0,C 180,E1 -7104.053,E2 -7104.053} C_VEL
LIN {X 0,Y 474.892,Z 134.329,A -85,B 0,C 180,E1 -7107.456,E2 -7107.456} C_VEL
LIN {X 0,Y 474.909,Z 134.324,A -85,B 0,C 180,E1 -7110,E2 -7110} C_VEL
LIN {X 0,Y 474.892,Z 134.329,A -85,B 0,C 180,E1 -7112.545,E2 -7112.545} C_VEL
LIN {X 0,Y 474.779,Z 134.34,A -85,B 0,C 180,E1 -7115.948,E2 -7115.948} C_VEL
LIN {X 0,Y 474.726,Z 134.35,A -85,B 0,C 180,E1 -7118.514,E2 -7118.514} C_VEL
LIN {X 0,Y 474.702,Z 134.35,A -85,B 0,C 180,E1 -7121.963,E2 -7121.963} C_VEL
LIN {X 0,Y 474.698,Z 134.354,A -85,B 0,C 180,E1 -7125.456,E2 -7125.456} C_VEL
LIN {X 0,Y 474.724,Z 134.495,A -85,B 0,C 180,E1 -7128.058,E2 -7128.058} C_VEL
LIN {X 0,Y 475.627,Z 140.778,A -85,B 0,C 180,E1 -7129.419,E2 -7129.419} C_VEL
LIN {X 0,Y 475.48,Z 150.176,A -85,B 0,C 180,E1 -7131.336,E2 -7131.336} C_VEL
LIN {X 0,Y 478.179,Z 163.476,A -85,B 0,C 180,E1 -7131.643,E2 -7131.643} C_VEL
LIN {X 0,Y 477.337,Z 257.318,A -85,B 0,C 180,E1 -7133.109,E2 -7133.109} C_VEL
LIN {X 0,Y 477.068,Z 270.734,A -85,B 0,C 180,E1 -7133.496,E2 -7133.496} C_VEL
LIN {X 0,Y 476.802,Z 283.412,A -85,B 0,C 180,E1 -7134.041,E2 -7134.041} C_VEL
LIN {X 0,Y 476.426,Z 295.423,A -85,B 0,C 180,E1 -7134.745,E2 -7134.745} C_VEL
LIN {X 0,Y 475.905,Z 306.974,A -85,B 0,C 180,E1 -7135.613,E2 -7135.613} C_VEL
LIN {X 0,Y 475.485,Z 317.022,A -85,B 0,C 180,E1 -7136.559,E2 -7136.559} C_VEL
LIN {X 0,Y 475.098,Z 325.779,A -85,B 0,C 180,E1 -7137.572,E2 -7137.572} C_VEL
LIN {X 0,Y 474.748,Z 334.173,A -85,B 0,C 180,E1 -7138.759,E2 -7138.759} C_VEL
LIN {X 0,Y 474.43,Z 341.303,A -85,B 0,C 180,E1 -7139.998,E2 -7139.998} C_VEL
LIN {X 0,Y 474.193,Z 347.108,A -85,B 0,C 180,E1 -7141.248,E2 -7141.248} C_VEL
LIN {X 0,Y 473.967,Z 352.588,A -85,B 0,C 180,E1 -7142.767,E2 -7142.767} C_VEL
LIN {X 0,Y 473.814,Z 356.558,A -85,B 0,C 180,E1 -7144.309,E2 -7144.309} C_VEL
LIN {X 0,Y 473.711,Z 358.47,A -85,B 0,C 180,E1 -7145.353,E2 -7145.353} C_VEL
LIN {X 0,Y 473.668,Z 360.022,A -85,B 0,C 180,E1 -7146.754,E2 -7146.754} C_VEL
LIN {X 0,Y 473.647,Z 360.495,A -85,B 0,C 180,E1 -7148.149,E2 -7148.149} C_VEL
LIN {X 0,Y 473.663,Z 359.809,A -85,B 0,C 180,E1 -7149.645,E2 -7149.645} C_VEL
LIN {X 0,Y 473.761,Z 358.399,A -85,B 0,C 180,E1 -7150.839,E2 -7150.839} C_VEL
LIN {X 0,Y 473.929,Z 354.937,A -85,B 0,C 180,E1 -7152.539,E2 -7152.539} C_VEL
LIN {X 0,Y 474.026,Z 351.376,A -85,B 0,C 180,E1 -7153.756,E2 -7153.756} C_VEL
LIN {X 0,Y 474.21,Z 346.858,A -85,B 0,C 180,E1 -7154.961,E2 -7154.961} C_VEL
LIN {X 0,Y 474.475,Z 341.251,A -85,B 0,C 180,E1 -7156.16,E2 -7156.16} C_VEL
LIN {X 0,Y 474.77,Z 333.877,A -85,B 0,C 180,E1 -7157.437,E2 -7157.437} C_VEL
LIN {X 0,Y 475.175,Z 325.259,A -85,B 0,C 180,E1 -7158.641,E2 -7158.641} C_VEL
LIN {X 0,Y 475.649,Z 315.43,A -85,B 0,C 180,E1 -7159.744,E2 -7159.744} C_VEL
LIN {X 0,Y 476.011,Z 304.962,A -85,B 0,C 180,E1 -7160.697,E2 -7160.697} C_VEL
LIN {X 0,Y 476.587,Z 293.908,A -85,B 0,C 180,E1 -7161.495,E2 -7161.495} C_VEL
LIN {X 0,Y 476.952,Z 282.52,A -85,B 0,C 180,E1 -7162.137,E2 -7162.137} C_VEL
LIN {X 0,Y 477.208,Z 269.452,A -85,B 0,C 180,E1 -7162.682,E2 -7162.682} C_VEL
LIN {X 0,Y 477.461,Z 256.23,A -85,B 0,C 180,E1 -7163.043,E2 -7163.043} C_VEL
LIN {X 0,Y 478.173,Z 162.899,A -85,B 0,C 180,E1 -7164.508,E2 -7164.508} C_VEL
LIN {X 0,Y 475.565,Z 150.389,A -85,B 0,C 180,E1 -7164.823,E2 -7164.823} C_VEL
LIN {X 0,Y 475.662,Z 140.259,A -85,B 0,C 180,E1 -7166.861,E2 -7166.861} C_VEL
LIN {X 0,Y 474.661,Z 134.362,A -85,B 0,C 180,E1 -7168.103,E2 -7168.103} C_VEL
LIN {X 0,Y 474.645,Z 134.363,A -85,B 0,C 180,E1 -7171.718,E2 -7171.718} C_VEL
LIN {X 0,Y 474.653,Z 134.362,A -85,B 0,C 180,E1 -7174.584,E2 -7174.584} C_VEL
LIN {X 0,Y 474.603,Z 134.37,A -85,B 0,C 180,E1 -7177.356,E2 -7177.356} C_VEL
LIN {X 0,Y 474.656,Z 134.358,A -85,B 0,C 180,E1 -7180.09,E2 -7180.09} C_VEL
LIN {X 0,Y 474.638,Z 134.364,A -85,B 0,C 180,E1 -7182.775,E2 -7182.775} C_VEL
LIN {X 0,Y 474.647,Z 134.361,A -85,B 0,C 180,E1 -7185.421,E2 -7185.421} C_VEL
LIN {X 0,Y 474.709,Z 134.353,A -85,B 0,C 180,E1 -7188.038,E2 -7188.038} C_VEL
LIN {X 0,Y 474.712,Z 134.352,A -85,B 0,C 180,E1 -7191.487,E2 -7191.487} C_VEL
LIN {X 0,Y 474.744,Z 134.35,A -85,B 0,C 180,E1 -7194.052,E2 -7194.052} C_VEL
LIN {X 0,Y 474.878,Z 134.33,A -85,B 0,C 180,E1 -7197.456,E2 -7197.456} C_VEL
LIN {X 0,Y 474.884,Z 134.329,A -85,B 0,C 180,E1 -7200,E2 -7200} C_VEL
LIN {X 0,Y 474.875,Z 134.328,A -85,B 0,C 180,E1 -7202.545,E2 -7202.545} C_VEL
LIN {X 0,Y 474.74,Z 134.35,A -85,B 0,C 180,E1 -7205.949,E2 -7205.949} C_VEL
LIN {X 0,Y 474.665,Z 134.356,A -85,B 0,C 180,E1 -7208.515,E2 -7208.515} C_VEL
LIN {X 0,Y 474.689,Z 134.356,A -85,B 0,C 180,E1 -7211.963,E2 -7211.963} C_VEL
LIN {X 0,Y 474.655,Z 134.357,A -85,B 0,C 180,E1 -7215.458,E2 -7215.458} C_VEL
LIN {X 0,Y 474.583,Z 134.365,A -85,B 0,C 180,E1 -7219.014,E2 -7219.014} C_VEL
LIN {X 0,Y 474.574,Z 134.37,A -85,B 0,C 180,E1 -7221.73,E2 -7221.73} C_VEL
LIN {X 0,Y 474.587,Z 134.363,A -85,B 0,C 180,E1 -7224.497,E2 -7224.497} C_VEL
LIN {X 0,Y 474.597,Z 134.366,A -85,B 0,C 180,E1 -7227.327,E2 -7227.327} C_VEL
LIN {X 0,Y 474.554,Z 134.369,A -85,B 0,C 180,E1 -7230.234,E2 -7230.234} C_VEL
LIN {X 0,Y 474.619,Z 134.366,A -85,B 0,C 180,E1 -7233.222,E2 -7233.222} C_VEL
LIN {X 0,Y 474.588,Z 134.365,A -85,B 0,C 180,E1 -7236.324,E2 -7236.324} C_VEL
LIN {X 0,Y 474.627,Z 134.361,A -85,B 0,C 180,E1 -7239.548,E2 -7239.548} C_VEL
LIN {X 0,Y 474.581,Z 134.368,A -85,B 0,C 180,E1 -7242.23,E2 -7242.23} C_VEL
LIN {X 0,Y 474.621,Z 134.364,A -85,B 0,C 180,E1 -7245.298,E2 -7245.298} C_VEL
LIN {X 0,Y 474.61,Z 134.369,A -85,B 0,C 180,E1 -7248.213,E2 -7248.213} C_VEL
LIN {X 0,Y 474.613,Z 134.363,A -85,B 0,C 180,E1 -7251.542,E2 -7251.542} C_VEL
LIN {X 0,Y 474.627,Z 134.363,A -85,B 0,C 180,E1 -7254.725,E2 -7254.725} C_VEL
LIN {X 0,Y 474.64,Z 134.366,A -85,B 0,C 180,E1 -7257.787,E2 -7257.787} C_VEL
LIN {X 0,Y 474.612,Z 134.364,A -85,B 0,C 180,E1 -7260.888,E2 -7260.888} C_VEL
LIN {X 0,Y 474.689,Z 134.501,A -85,B 0,C 180,E1 -7263.881,E2 -7263.881} C_VEL
LIN {X 0,Y 476.555,Z 144.058,A -85,B 0,C 180,E1 -7265.61,E2 -7265.61} C_VEL
LIN {X 0,Y 476.724,Z 148.456,A -85,B 0,C 180,E1 -7266.362,E2 -7266.362} C_VEL
LIN {X 0,Y 476.002,Z 165.865,A -85,B 0,C 180,E1 -7269.246,E2 -7269.246} C_VEL
LIN {X 0,Y 475.423,Z 183.508,A -85,B 0,C 180,E1 -7272.137,E2 -7272.137} C_VEL
LIN {X 0,Y 475.242,Z 190.282,A -85,B 0,C 180,E1 -7273.21,E2 -7273.21} C_VEL
LIN {X 0,Y 477.998,Z 210.044,A -85,B 0,C 180,E1 -7273.627,E2 -7273.627} C_VEL
LIN {X 0,Y 477.299,Z 299.761,A -85,B 0,C 180,E1 -7275.04,E2 -7275.04} C_VEL
LIN {X 0,Y 476.929,Z 312.695,A -85,B 0,C 180,E1 -7275.41,E2 -7275.41} C_VEL
LIN {X 0,Y 476.475,Z 324.721,A -85,B 0,C 180,E1 -7275.914,E2 -7275.914} C_VEL
LIN {X 0,Y 476.028,Z 336.113,A -85,B 0,C 180,E1 -7276.553,E2 -7276.553} C_VEL
LIN {X 0,Y 475.566,Z 347.907,A -85,B 0,C 180,E1 -7277.413,E2 -7277.413} C_VEL
LIN {X 0,Y 475.104,Z 358.44,A -85,B 0,C 180,E1 -7278.372,E2 -7278.372} C_VEL
LIN {X 0,Y 474.699,Z 367.091,A -85,B 0,C 180,E1 -7279.335,E2 -7279.335} C_VEL
LIN {X 0,Y 474.398,Z 375.077,A -85,B 0,C 180,E1 -7280.406,E2 -7280.406} C_VEL
LIN {X 0,Y 474.094,Z 382.883,A -85,B 0,C 180,E1 -7281.689,E2 -7281.689} C_VEL
LIN {X 0,Y 473.897,Z 390.074,A -85,B 0,C 180,E1 -7283.186,E2 -7283.186} C_VEL
LIN {X 0,Y 473.831,Z 394.868,A -85,B 0,C 180,E1 -7284.467,E2 -7284.467} C_VEL
LIN {X 0,Y 473.736,Z 398.532,A -85,B 0,C 180,E1 -7285.746,E2 -7285.746} C_VEL
LIN {X 0,Y 473.806,Z 400.429,A -85,B 0,C 180,E1 -7286.598,E2 -7286.598} C_VEL
LIN {X 0,Y 473.766,Z 401.849,A -85,B 0,C 180,E1 -7287.449,E2 -7287.449} C_VEL
LIN {X 0,Y 473.757,Z 402.866,A -85,B 0,C 180,E1 -7288.299,E2 -7288.299} C_VEL
LIN {X 0,Y 473.697,Z 403.488,A -85,B 0,C 180,E1 -7289.149,E2 -7289.149} C_VEL
LIN {X 0,Y 473.683,Z 403.713,A -85,B 0,C 180,E1 -7290,E2 -7290} C_VEL
LIN {X 0,Y 473.757,Z 402.895,A -85,B 0,C 180,E1 -7291.7,E2 -7291.7} C_VEL
LIN {X 0,Y 473.766,Z 401.895,A -85,B 0,C 180,E1 -7292.55,E2 -7292.55} C_VEL
LIN {X 0,Y 473.806,Z 400.486,A -85,B 0,C 180,E1 -7293.401,E2 -7293.401} C_VEL
LIN {X 0,Y 473.76,Z 397.52,A -85,B 0,C 180,E1 -7294.679,E2 -7294.679} C_VEL
LIN {X 0,Y 473.81,Z 393.503,A -85,B 0,C 180,E1 -7295.959,E2 -7295.959} C_VEL
LIN {X 0,Y 473.999,Z 387.318,A -85,B 0,C 180,E1 -7297.454,E2 -7297.454} C_VEL
LIN {X 0,Y 474.182,Z 380.564,A -85,B 0,C 180,E1 -7298.738,E2 -7298.738} C_VEL
LIN {X 0,Y 474.468,Z 372.183,A -85,B 0,C 180,E1 -7300.023,E2 -7300.023} C_VEL
LIN {X 0,Y 474.893,Z 363.56,A -85,B 0,C 180,E1 -7301.092,E2 -7301.092} C_VEL
LIN {X 0,Y 475.318,Z 353.37,A -85,B 0,C 180,E1 -7302.122,E2 -7302.122} C_VEL
LIN {X 0,Y 475.761,Z 342.379,A -85,B 0,C 180,E1 -7303.019,E2 -7303.019} C_VEL
LIN {X 0,Y 476.251,Z 330.744,A -85,B 0,C 180,E1 -7303.765,E2 -7303.765} C_VEL
LIN {X 0,Y 476.668,Z 318.666,A -85,B 0,C 180,E1 -7304.352,E2 -7304.352} C_VEL
LIN {X 0,Y 477.105,Z 305.597,A -85,B 0,C 180,E1 -7304.802,E2 -7304.802} C_VEL
LIN {X 0,Y 477.323,Z 293.221,A -85,B 0,C 180,E1 -7305.068,E2 -7305.068} C_VEL
LIN {X 0,Y 477.903,Z 209.358,A -85,B 0,C 180,E1 -7306.361,E2 -7306.361} C_VEL
LIN {X 0,Y 475.25,Z 190.698,A -85,B 0,C 180,E1 -7306.76,E2 -7306.76} C_VEL
LIN {X 0,Y 475.876,Z 171.895,A -85,B 0,C 180,E1 -7309.857,E2 -7309.857} C_VEL
LIN {X 0,Y 476.699,Z 153.064,A -85,B 0,C 180,E1 -7312.997,E2 -7312.997} C_VEL
LIN {X 0,Y 476.962,Z 146.44,A -85,B 0,C 180,E1 -7314.116,E2 -7314.116} C_VEL
LIN {X 0,Y 474.691,Z 134.358,A -85,B 0,C 180,E1 -7316.317,E2 -7316.317} C_VEL
LIN {X 0,Y 474.621,Z 134.363,A -85,B 0,C 180,E1 -7319.251,E2 -7319.251} C_VEL
LIN {X 0,Y 474.616,Z 134.365,A -85,B 0,C 180,E1 -7322.43,E2 -7322.43} C_VEL
LIN {X 0,Y 474.615,Z 134.362,A -85,B 0,C 180,E1 -7325.469,E2 -7325.469} C_VEL
LIN {X 0,Y 474.612,Z 134.362,A -85,B 0,C 180,E1 -7328.457,E2 -7328.457} C_VEL
LIN {X 0,Y 474.628,Z 134.359,A -85,B 0,C 180,E1 -7330.959,E2 -7330.959} C_VEL
LIN {X 0,Y 474.605,Z 134.365,A -85,B 0,C 180,E1 -7334.105,E2 -7334.105} C_VEL
LIN {X 0,Y 474.614,Z 134.361,A -85,B 0,C 180,E1 -7337.065,E2 -7337.065} C_VEL
LIN {X 0,Y 474.617,Z 134.361,A -85,B 0,C 180,E1 -7340.353,E2 -7340.353} C_VEL
LIN {X 0,Y 474.588,Z 134.371,A -85,B 0,C 180,E1 -7343.676,E2 -7343.676} C_VEL
LIN {X 0,Y 474.624,Z 134.36,A -85,B 0,C 180,E1 -7346.778,E2 -7346.778} C_VEL
LIN {X 0,Y 474.604,Z 134.366,A -85,B 0,C 180,E1 -7349.769,E2 -7349.769} C_VEL
LIN {X 0,Y 474.696,Z 134.351,A -85,B 0,C 180,E1 -7352.679,E2 -7352.679} C_VEL
LIN {X 0,Y 474.656,Z 134.361,A -85,B 0,C 180,E1 -7355.507,E2 -7355.507} C_VEL
LIN {X 0,Y 474.669,Z 134.361,A -85,B 0,C 180,E1 -7359.185,E2 -7359.185} C_VEL
LIN {X 0,Y 474.645,Z 134.357,A -85,B 0,C 180,E1 -7361.883,E2 -7361.883} C_VEL
LIN {X 0,Y 474.698,Z 134.351,A -85,B 0,C 180,E1 -7364.544,E2 -7364.544} C_VEL
LIN {X 0,Y 474.703,Z 134.349,A -85,B 0,C 180,E1 -7368.037,E2 -7368.037} C_VEL
LIN {X 0,Y 474.726,Z 134.349,A -85,B 0,C 180,E1 -7371.486,E2 -7371.486} C_VEL
LIN {X 0,Y 474.77,Z 134.341,A -85,B 0,C 180,E1 -7374.052,E2 -7374.052} C_VEL
LIN {X 0,Y 474.893,Z 134.327,A -85,B 0,C 180,E1 -7377.455,E2 -7377.455} C_VEL
LIN {X 0,Y 474.91,Z 134.324,A -85,B 0,C 180,E1 -7380,E2 -7380} C_VEL
LIN {X 0,Y 474.893,Z 134.331,A -85,B 0,C 180,E1 -7382.544,E2 -7382.544} C_VEL
LIN {X 0,Y 474.769,Z 134.341,A -85,B 0,C 180,E1 -7385.947,E2 -7385.947} C_VEL
LIN {X 0,Y 474.726,Z 134.353,A -85,B 0,C 180,E1 -7388.513,E2 -7388.513} C_VEL
LIN {X 0,Y 474.702,Z 134.351,A -85,B 0,C 180,E1 -7391.962,E2 -7391.962} C_VEL
LIN {X 0,Y 474.698,Z 134.35,A -85,B 0,C 180,E1 -7395.455,E2 -7395.455} C_VEL
LIN {X 0,Y 474.662,Z 134.356,A -85,B 0,C 180,E1 -7399.01,E2 -7399.01} C_VEL
LIN {X 0,Y 474.585,Z 134.365,A -85,B 0,C 180,E1 -7401.729,E2 -7401.729} C_VEL
LIN {X 0,Y 474.654,Z 134.362,A -85,B 0,C 180,E1 -7404.493,E2 -7404.493} C_VEL
LIN {X 0,Y 474.695,Z 134.35,A -85,B 0,C 180,E1 -7407.338,E2 -7407.338} C_VEL
LIN {X 0,Y 474.601,Z 134.363,A -85,B 0,C 180,E1 -7410.81,E2 -7410.81} C_VEL
LIN {X 0,Y 474.634,Z 134.364,A -85,B 0,C 180,E1 -7413.984,E2 -7413.984} C_VEL
LIN {X 0,Y 474.571,Z 134.366,A -85,B 0,C 180,E1 -7416.9,E2 -7416.9} C_VEL
LIN {X 0,Y 474.65,Z 134.359,A -85,B 0,C 180,E1 -7419.652,E2 -7419.652} C_VEL
LIN {X 0,Y 474.647,Z 134.356,A -85,B 0,C 180,E1 -7422.93,E2 -7422.93} C_VEL
LIN {X 0,Y 474.613,Z 134.369,A -85,B 0,C 180,E1 -7425.896,E2 -7425.896} C_VEL
LIN {X 0,Y 474.641,Z 134.357,A -85,B 0,C 180,E1 -7429.038,E2 -7429.038} C_VEL
LIN {X 0,Y 474.615,Z 134.367,A -85,B 0,C 180,E1 -7431.702,E2 -7431.702} C_VEL
LIN {X 0,Y 474.624,Z 134.359,A -85,B 0,C 180,E1 -7434.726,E2 -7434.726} C_VEL
LIN {X 0,Y 474.633,Z 134.365,A -85,B 0,C 180,E1 -7437.788,E2 -7437.788} C_VEL
LIN {X 0,Y 474.619,Z 134.36,A -85,B 0,C 180,E1 -7440.885,E2 -7440.885} C_VEL
LIN {X 0,Y 474.662,Z 134.361,A -85,B 0,C 180,E1 -7443.629,E2 -7443.629} C_VEL
LIN {X 0,Y 474.631,Z 134.358,A -85,B 0,C 180,E1 -7446.641,E2 -7446.641} C_VEL
LIN {X 0,Y 474.652,Z 134.356,A -85,B 0,C 180,E1 -7450.09,E2 -7450.09} C_VEL
LIN {X 0,Y 474.651,Z 134.36,A -85,B 0,C 180,E1 -7451.672,E2 -7451.672} C_VEL
LIN {X 0,Y 473.988,Z 134.439,A -85,B 0,C 180,E1 -7452.381,E2 -7452.381} C_VEL
LIN {X 0,Y 471.139,Z 134.799,A -85,B 0,C 180,E1 -7453.533,E2 -7453.533} C_VEL
LIN {X 0,Y 468.724,Z 135.103,A -85,B 0,C 180,E1 -7454.461,E2 -7454.461} C_VEL
LIN {X 0,Y 467.683,Z 135.23,A -85,B 0,C 180,E1 -7455.178,E2 -7455.178} C_VEL
LIN {X 0,Y 467.596,Z 135.238,A -85,B 0,C 180,E1 -7455.421,E2 -7455.421} C_VEL
LIN {X 0,Y 467.65,Z 135.23,A -85,B 0,C 180,E1 -7458.734,E2 -7458.734} C_VEL
LIN {X 0,Y 467.745,Z 135.216,A -85,B 0,C 180,E1 -7462.229,E2 -7462.229} C_VEL
LIN {X 0,Y 467.723,Z 135.223,A -85,B 0,C 180,E1 -7464.828,E2 -7464.828} C_VEL
LIN {X 0,Y 467.857,Z 135.206,A -85,B 0,C 180,E1 -7467.418,E2 -7467.418} C_VEL
LIN {X 0,Y 467.88,Z 135.199,A -85,B 0,C 180,E1 -7470,E2 -7470} C_VEL
LIN {X 0,Y 467.857,Z 135.205,A -85,B 0,C 180,E1 -7472.583,E2 -7472.583} C_VEL
LIN {X 0,Y 467.743,Z 135.216,A -85,B 0,C 180,E1 -7476.038,E2 -7476.038} C_VEL
LIN {X 0,Y 467.679,Z 135.23,A -85,B 0,C 180,E1 -7478.643,E2 -7478.643} C_VEL
LIN {X 0,Y 467.653,Z 135.229,A -85,B 0,C 180,E1 -7482.146,E2 -7482.146} C_VEL
LIN {X 0,Y 467.65,Z 135.232,A -85,B 0,C 180,E1 -7485.695,E2 -7485.695} C_VEL
LIN {X 0,Y 467.65,Z 135.327,A -85,B 0,C 180,E1 -7487.888,E2 -7487.888} C_VEL
LIN {X 0,Y 468.631,Z 141.586,A -85,B 0,C 180,E1 -7489.265,E2 -7489.265} C_VEL
LIN {X 0,Y 468.516,Z 150.229,A -85,B 0,C 180,E1 -7491.073,E2 -7491.073} C_VEL
LIN {X 0,Y 471.375,Z 165.207,A -85,B 0,C 180,E1 -7491.43,E2 -7491.43} C_VEL
LIN {X 0,Y 470.453,Z 257.777,A -85,B 0,C 180,E1 -7492.9,E2 -7492.9} C_VEL
LIN {X 0,Y 470.201,Z 271.477,A -85,B 0,C 180,E1 -7493.305,E2 -7493.305} C_VEL
LIN {X 0,Y 469.905,Z 283.238,A -85,B 0,C 180,E1 -7493.818,E2 -7493.818} C_VEL
LIN {X 0,Y 469.559,Z 294.859,A -85,B 0,C 180,E1 -7494.497,E2 -7494.497} C_VEL
LIN {X 0,Y 469.079,Z 305.386,A -85,B 0,C 180,E1 -7495.278,E2 -7495.278} C_VEL
LIN {X 0,Y 468.561,Z 316.205,A -85,B 0,C 180,E1 -7496.28,E2 -7496.28} C_VEL
LIN {X 0,Y 468.186,Z 324.703,A -85,B 0,C 180,E1 -7497.248,E2 -7497.248} C_VEL
LIN {X 0,Y 467.762,Z 333.645,A -85,B 0,C 180,E1 -7498.493,E2 -7498.493} C_VEL
LIN {X 0,Y 467.45,Z 340.901,A -85,B 0,C 180,E1 -7499.746,E2 -7499.746} C_VEL
LIN {X 0,Y 467.182,Z 346.646,A -85,B 0,C 180,E1 -7500.967,E2 -7500.967} C_VEL
LIN {X 0,Y 466.938,Z 352.483,A -85,B 0,C 180,E1 -7502.557,E2 -7502.557} C_VEL
LIN {X 0,Y 466.753,Z 356.53,A -85,B 0,C 180,E1 -7504.092,E2 -7504.092} C_VEL
LIN {X 0,Y 466.598,Z 359.13,A -85,B 0,C 180,E1 -7505.576,E2 -7505.576} C_VEL
LIN {X 0,Y 466.577,Z 360.521,A -85,B 0,C 180,E1 -7507.051,E2 -7507.051} C_VEL
LIN {X 0,Y 466.565,Z 360.771,A -85,B 0,C 180,E1 -7508.438,E2 -7508.438} C_VEL
LIN {X 0,Y 466.588,Z 360.012,A -85,B 0,C 180,E1 -7509.809,E2 -7509.809} C_VEL
